(* CODESYS project cy-023_B_PLC1-ifm-206 (AF Logistic Principale).project

Project tree, tasks and I/O mapping:
  AC14nn : AC14nn, ifm electronic, order no. AC14nn, version 3.5.3.002
    application Application
      libraries: ACnnnn_Utils, * (ifm electronic); Standard, * (System); Util, * (System); SysRtc23, 3.4.0.0 (System); SysSocket23, 3.5.4.10 (System); SysFile, 3.5.6.0 (System); SysTypes Interfaces, * (System); CmpErrors Interfaces, * (System); VisuDialogs, * (System); SysFileAsync, 3.5.5.0 (System); NETWORK, 1.2.1.0 (OSCAT)
      task MainTask (cyclic, interval t#20ms, priority 15) calls PLC_PRG
      task EventTask (cyclic, interval t#20ms, priority 5) calls PLC_RT
      task VISU_TASK (cyclic, interval t#200ms, priority 30) calls VisuElems.Visu_Prg
      visualisation VIS_CHONOEDITOR
      visualisation PLC_FileManager
      visualisation PLC_Visualization
    ASi_Master_1 : ASi Master 1, ifm electronic, version 3.5.3.002
      ASi_1_binaryIO : ASi_1_binaryIO, ifm ecomatic gmbh, version 3.5.3.002
          input  Application.PSG_LIST[61] : BOOL  // ASi Input bin.Digital S(A) Slave.Digital S(A) Slave.Bit0
          input  Application.PSG_LIST[62] : BOOL  // ASi Input bin.Digital S(A) Slave.Digital S(A) Slave.Bit2
          input  Application.PSG_LIST[63] : BOOL  // ASi Input bin.Digital S(A) Slave.Digital S(A) Slave.Bit0
          input  Application.PSG_LIST[64] : BOOL  // ASi Input bin.Digital S(A) Slave.Digital S(A) Slave.Bit2
          input  Application.PSG_LIST[65] : BOOL  // ASi Input bin.Digital S(A) Slave.Digital S(A) Slave.Bit0
          input  Application.PSG_LIST[66] : BOOL  // ASi Input bin.Digital S(A) Slave.Digital S(A) Slave.Bit2
          input  Application.PSG_LIST[67] : BOOL  // ASi Input bin.Digital S(A) Slave.Digital S(A) Slave.Bit0
          input  Application.PSG_LIST[68] : BOOL  // ASi Input bin.Digital S(A) Slave.Digital S(A) Slave.Bit2
          input  Application.PSG_LIST[69] : BOOL  // ASi Input bin.Digital S(A) Slave.Digital S(A) Slave.Bit0
          input  Application.PSG_LIST[70] : BOOL  // ASi Input bin.Digital S(A) Slave.Digital S(A) Slave.Bit2
          input  Application.PSG_LIST[71] : BOOL  // ASi Input bin.Digital S(A) Slave.Digital S(A) Slave.Bit0
          input  Application.PSG_LIST[72] : BOOL  // ASi Input bin.Digital S(A) Slave.Digital S(A) Slave.Bit2
          input  Application.PSG_LIST[73] : BOOL  // ASi Input bin.Digital S(A) Slave.Digital S(A) Slave.Bit0
          input  Application.PSG_LIST[74] : BOOL  // ASi Input bin.Digital S(A) Slave.Digital S(A) Slave.Bit2
          input  Application.PSG_LIST[75] : BOOL  // ASi Input bin.Digital S(A) Slave.Digital S(A) Slave.Bit0
          input  Application.PSG_LIST[76] : BOOL  // ASi Input bin.Digital S(A) Slave.Digital S(A) Slave.Bit2
          input  Application.PSG_LIST[77] : BOOL  // ASi Input bin.Digital S(A) Slave.Digital S(A) Slave.Bit0
          input  Application.PSG_LIST[78] : BOOL  // ASi Input bin.Digital S(A) Slave.Digital S(A) Slave.Bit2
          input  Application.PSG_LIST[79] : BOOL  // ASi Input bin.Digital S(A) Slave.Digital S(A) Slave.Bit0
          input  Application.PSG_LIST[80] : BOOL  // ASi Input bin.Digital S(A) Slave.Digital S(A) Slave.Bit2
          input  Application.PSG_LIST[81] : BOOL  // ASi Input bin.Digital S(A) Slave.Digital S(A) Slave.Bit0
          input  Application.PSG_LIST[82] : BOOL  // ASi Input bin.Digital S(A) Slave.Digital S(A) Slave.Bit2
          input  Application.PSG_LIST[83] : BOOL  // ASi Input bin.Digital S(A) Slave.Digital S(A) Slave.Bit0
          input  Application.PSG_LIST[84] : BOOL  // ASi Input bin.Digital S(A) Slave.Digital S(A) Slave.Bit2
          input  Application.PSG_LIST[85] : BOOL  // ASi Input bin.Digital S(A) Slave.Digital S(A) Slave.Bit0
          input  Application.PSG_LIST[86] : BOOL  // ASi Input bin.Digital S(A) Slave.Digital S(A) Slave.Bit2
          input  Application.PSG_LIST[87] : BOOL  // ASi Input bin.Digital S(A) Slave.Digital S(A) Slave.Bit0
          input  Application.PSG_LIST[88] : BOOL  // ASi Input bin.Digital S(A) Slave.Digital S(A) Slave.Bit2
          input  Application.PSG_LIST[121] : BOOL  // ASi Input bin.Digital S(A) Slave.Digital S(A) Slave.Bit0
          input  Application.PSG_LIST[122] : BOOL  // ASi Input bin.Digital S(A) Slave.Digital S(A) Slave.Bit2
          input  Application.PSG_LIST[123] : BOOL  // ASi Input bin.Digital S(A) Slave.Digital S(A) Slave.Bit0
          input  Application.PSG_LIST[124] : BOOL  // ASi Input bin.Digital S(A) Slave.Digital S(A) Slave.Bit2
          input  Application.PSG_LIST[125] : BOOL  // ASi Input bin.Digital S(A) Slave.Digital S(A) Slave.Bit0
          input  Application.PSG_LIST[126] : BOOL  // ASi Input bin.Digital S(A) Slave.Digital S(A) Slave.Bit2
          input  Application.PSG_LIST[127] : BOOL  // ASi Input bin.Digital S(A) Slave.Digital S(A) Slave.Bit0
          input  Application.PSG_LIST[128] : BOOL  // ASi Input bin.Digital S(A) Slave.Digital S(A) Slave.Bit2
          input  Application.PSG_LIST[129] : BOOL  // ASi Input bin.Digital S(A) Slave.Digital S(A) Slave.Bit0
          input  Application.PSG_LIST[130] : BOOL  // ASi Input bin.Digital S(A) Slave.Digital S(A) Slave.Bit2
          input  Application.PSG_LIST[131] : BOOL  // ASi Input bin.Digital S(A) Slave.Digital S(A) Slave.Bit0
          input  Application.PSG_LIST[132] : BOOL  // ASi Input bin.Digital S(A) Slave.Digital S(A) Slave.Bit2
          input  Application.PSG_LIST[133] : BOOL  // ASi Input bin.Digital S(A) Slave.Digital S(A) Slave.Bit0
          input  Application.PSG_LIST[134] : BOOL  // ASi Input bin.Digital S(A) Slave.Digital S(A) Slave.Bit2
          input  Application.PSG_LIST[135] : BOOL  // ASi Input bin.Digital S(A) Slave.Digital S(A) Slave.Bit0
          input  Application.PSG_LIST[136] : BOOL  // ASi Input bin.Digital S(A) Slave.Digital S(A) Slave.Bit2
          input  Application.PSG_LIST[137] : BOOL  // ASi Input bin.Digital S(A) Slave.Digital S(A) Slave.Bit0
          input  Application.PSG_LIST[138] : BOOL  // ASi Input bin.Digital S(A) Slave.Digital S(A) Slave.Bit2
          input  Application.PSG_LIST[139] : BOOL  // ASi Input bin.Digital S(A) Slave.Digital S(A) Slave.Bit0
          input  Application.PSG_LIST[140] : BOOL  // ASi Input bin.Digital S(A) Slave.Digital S(A) Slave.Bit2
          input  Application.PSG_LIST[141] : BOOL  // ASi Input bin.Digital S(A) Slave.Digital S(A) Slave.Bit0
          input  Application.PSG_LIST[142] : BOOL  // ASi Input bin.Digital S(A) Slave.Digital S(A) Slave.Bit2
          input  Application.PSG_LIST[143] : BOOL  // ASi Input bin.Digital S(A) Slave.Digital S(A) Slave.Bit0
          input  Application.PSG_LIST[144] : BOOL  // ASi Input bin.Digital S(A) Slave.Digital S(A) Slave.Bit2
          input  Application.PSG_LIST[145] : BOOL  // ASi Input bin.Digital S(A) Slave.Digital S(A) Slave.Bit0
          input  Application.PSG_LIST[146] : BOOL  // ASi Input bin.Digital S(A) Slave.Digital S(A) Slave.Bit2
          input  Application.PSG_LIST[147] : BOOL  // ASi Input bin.Digital S(A) Slave.Digital S(A) Slave.Bit0
          input  Application.PSG_LIST[148] : BOOL  // ASi Input bin.Digital S(A) Slave.Digital S(A) Slave.Bit2
          input  Application.LUX_ST[43] : BOOL  // ASi Input bin.Digital S(A) Slave.Digital S(A) Slave.Bit0
          input  Application.PSG_LIST[174] : BOOL  // ASi Input bin.Digital S(A) Slave.Digital S(A) Slave.Bit2
          input  Application.LUX_ST[44] : BOOL  // ASi Input bin.Digital S(A) Slave.Digital S(A) Slave.Bit0
          input  Application.PSG_LIST[176] : BOOL  // ASi Input bin.Digital S(A) Slave.Digital S(A) Slave.Bit2
          input  Application.LUX_ST[45] : BOOL  // ASi Input bin.Digital S(A) Slave.Digital S(A) Slave.Bit0
          input  Application.PSG_LIST[178] : BOOL  // ASi Input bin.Digital S(A) Slave.Digital S(A) Slave.Bit2
          input  Application.PSG_LIST[179] : BOOL  // ASi Input bin.Digital B Slave.Digital B Slave.Bit0
          input  Application.PSG_LIST[180] : BOOL  // ASi Input bin.Digital B Slave.Digital B Slave.Bit2
          input  Application.LUX_ST[46] : BOOL  // ASi Input bin.Digital B Slave.Digital B Slave.Bit0
          input  Application.LUX_ST[47] : BOOL  // ASi Input bin.Digital B Slave.Digital B Slave.Bit0
          input  Application.LUX_ST[48] : BOOL  // ASi Input bin.Digital B Slave.Digital B Slave.Bit0
          output Application.LUX_LIST[43] : BOOL  // ASi Output bin.Digital S(A) Slave.Digital S(A) Slave.Bit0
          output Application.LUX_LIST[44] : BOOL  // ASi Output bin.Digital S(A) Slave.Digital S(A) Slave.Bit0
          output Application.LUX_LIST[45] : BOOL  // ASi Output bin.Digital S(A) Slave.Digital S(A) Slave.Bit0
          output Application.LUX_LIST[46] : BOOL  // ASi Output bin.Digital B Slave.Digital B Slave.Bit0
          output Application.LUX_LIST[47] : BOOL  // ASi Output bin.Digital B Slave.Digital B Slave.Bit0
          output Application.LUX_LIST[48] : BOOL  // ASi Output bin.Digital B Slave.Digital B Slave.Bit0
          unmapped channels: ASi Input bin, ASi Output bin
      ASi_1_analogIO : ASi_1_analogIO, ifm ecomatic gmbh, version 3.5.3.002
          unmapped channels: ASi Input, ASi Output
    ASi_Master_2 : ASi Master 2, ifm electronic, version 3.5.3.002
      ASi_2_binaryIO : ASi_2_binaryIO, ifm ecomatic gmbh, version 3.5.3.002
          input  Application.PSG_LIST[1] : BOOL  // ASi Input bin.Digital S(A) Slave.Digital S(A) Slave.Bit0
          input  Application.PSG_LIST[2] : BOOL  // ASi Input bin.Digital S(A) Slave.Digital S(A) Slave.Bit2
          input  Application.PSG_LIST[3] : BOOL  // ASi Input bin.Digital S(A) Slave.Digital S(A) Slave.Bit0
          input  Application.PSG_LIST[4] : BOOL  // ASi Input bin.Digital S(A) Slave.Digital S(A) Slave.Bit2
          input  Application.PSG_LIST[5] : BOOL  // ASi Input bin.Digital S(A) Slave.Digital S(A) Slave.Bit0
          input  Application.PSG_LIST[6] : BOOL  // ASi Input bin.Digital S(A) Slave.Digital S(A) Slave.Bit2
          input  Application.PSG_LIST[7] : BOOL  // ASi Input bin.Digital S(A) Slave.Digital S(A) Slave.Bit0
          input  Application.PSG_LIST[8] : BOOL  // ASi Input bin.Digital S(A) Slave.Digital S(A) Slave.Bit2
          input  Application.PSG_LIST[9] : BOOL  // ASi Input bin.Digital S(A) Slave.Digital S(A) Slave.Bit0
          input  Application.PSG_LIST[10] : BOOL  // ASi Input bin.Digital S(A) Slave.Digital S(A) Slave.Bit2
          input  Application.PSG_LIST[11] : BOOL  // ASi Input bin.Digital S(A) Slave.Digital S(A) Slave.Bit0
          input  Application.PSG_LIST[12] : BOOL  // ASi Input bin.Digital S(A) Slave.Digital S(A) Slave.Bit2
          input  Application.PSG_LIST[13] : BOOL  // ASi Input bin.Digital S(A) Slave.Digital S(A) Slave.Bit0
          input  Application.PSG_LIST[14] : BOOL  // ASi Input bin.Digital S(A) Slave.Digital S(A) Slave.Bit2
          input  Application.PSG_LIST[15] : BOOL  // ASi Input bin.Digital S(A) Slave.Digital S(A) Slave.Bit0
          input  Application.PSG_LIST[16] : BOOL  // ASi Input bin.Digital S(A) Slave.Digital S(A) Slave.Bit2
          input  Application.PSG_LIST[17] : BOOL  // ASi Input bin.Digital S(A) Slave.Digital S(A) Slave.Bit0
          input  Application.PSG_LIST[18] : BOOL  // ASi Input bin.Digital S(A) Slave.Digital S(A) Slave.Bit2
          input  Application.PSG_LIST[19] : BOOL  // ASi Input bin.Digital S(A) Slave.Digital S(A) Slave.Bit0
          input  Application.PSG_LIST[20] : BOOL  // ASi Input bin.Digital S(A) Slave.Digital S(A) Slave.Bit2
          input  Application.PSG_LIST[21] : BOOL  // ASi Input bin.Digital S(A) Slave.Digital S(A) Slave.Bit0
          input  Application.PSG_LIST[22] : BOOL  // ASi Input bin.Digital S(A) Slave.Digital S(A) Slave.Bit2
          input  Application.PSG_LIST[23] : BOOL  // ASi Input bin.Digital S(A) Slave.Digital S(A) Slave.Bit0
          input  Application.PSG_LIST[24] : BOOL  // ASi Input bin.Digital S(A) Slave.Digital S(A) Slave.Bit2
          input  Application.PSG_LIST[25] : BOOL  // ASi Input bin.Digital S(A) Slave.Digital S(A) Slave.Bit0
          input  Application.PSG_LIST[26] : BOOL  // ASi Input bin.Digital S(A) Slave.Digital S(A) Slave.Bit2
          input  Application.PSG_LIST[27] : BOOL  // ASi Input bin.Digital S(A) Slave.Digital S(A) Slave.Bit0
          input  Application.PSG_LIST[28] : BOOL  // ASi Input bin.Digital S(A) Slave.Digital S(A) Slave.Bit2
          input  Application.PSG_LIST[181] : BOOL  // ASi Input bin.Digital S(A) Slave.Digital S(A) Slave.Bit0
          input  Application.PSG_LIST[182] : BOOL  // ASi Input bin.Digital S(A) Slave.Digital S(A) Slave.Bit2
          input  Application.PSG_LIST[183] : BOOL  // ASi Input bin.Digital S(A) Slave.Digital S(A) Slave.Bit0
          input  Application.PSG_LIST[184] : BOOL  // ASi Input bin.Digital S(A) Slave.Digital S(A) Slave.Bit2
          input  Application.PSG_LIST[185] : BOOL  // ASi Input bin.Digital S(A) Slave.Digital S(A) Slave.Bit0
          input  Application.PSG_LIST[186] : BOOL  // ASi Input bin.Digital S(A) Slave.Digital S(A) Slave.Bit2
          input  Application.PSG_LIST[187] : BOOL  // ASi Input bin.Digital S(A) Slave.Digital S(A) Slave.Bit0
          input  Application.PSG_LIST[188] : BOOL  // ASi Input bin.Digital S(A) Slave.Digital S(A) Slave.Bit2
          input  Application.PSG_LIST[189] : BOOL  // ASi Input bin.Digital S(A) Slave.Digital S(A) Slave.Bit0
          input  Application.PSG_LIST[190] : BOOL  // ASi Input bin.Digital S(A) Slave.Digital S(A) Slave.Bit2
          input  Application.PSG_LIST[191] : BOOL  // ASi Input bin.Digital S(A) Slave.Digital S(A) Slave.Bit0
          input  Application.PSG_LIST[192] : BOOL  // ASi Input bin.Digital S(A) Slave.Digital S(A) Slave.Bit2
          input  Application.PSG_LIST[193] : BOOL  // ASi Input bin.Digital S(A) Slave.Digital S(A) Slave.Bit0
          input  Application.PSG_LIST[194] : BOOL  // ASi Input bin.Digital S(A) Slave.Digital S(A) Slave.Bit2
          input  Application.PSG_LIST[195] : BOOL  // ASi Input bin.Digital S(A) Slave.Digital S(A) Slave.Bit0
          input  Application.PSG_LIST[196] : BOOL  // ASi Input bin.Digital S(A) Slave.Digital S(A) Slave.Bit2
          input  Application.PSG_LIST[197] : BOOL  // ASi Input bin.Digital S(A) Slave.Digital S(A) Slave.Bit0
          input  Application.PSG_LIST[198] : BOOL  // ASi Input bin.Digital S(A) Slave.Digital S(A) Slave.Bit2
          input  Application.PSG_LIST[199] : BOOL  // ASi Input bin.Digital S(A) Slave.Digital S(A) Slave.Bit0
          input  Application.PSG_LIST[200] : BOOL  // ASi Input bin.Digital S(A) Slave.Digital S(A) Slave.Bit2
          input  Application.PSG_LIST[201] : BOOL  // ASi Input bin.Digital S(A) Slave.Digital S(A) Slave.Bit0
          input  Application.PSG_LIST[202] : BOOL  // ASi Input bin.Digital S(A) Slave.Digital S(A) Slave.Bit2
          input  Application.PSG_LIST[203] : BOOL  // ASi Input bin.Digital S(A) Slave.Digital S(A) Slave.Bit0
          input  Application.PSG_LIST[204] : BOOL  // ASi Input bin.Digital S(A) Slave.Digital S(A) Slave.Bit2
          input  Application.PSG_LIST[205] : BOOL  // ASi Input bin.Digital S(A) Slave.Digital S(A) Slave.Bit0
          input  Application.PSG_LIST[206] : BOOL  // ASi Input bin.Digital S(A) Slave.Digital S(A) Slave.Bit2
          input  Application.PSG_LIST[207] : BOOL  // ASi Input bin.Digital S(A) Slave.Digital S(A) Slave.Bit0
          input  Application.PSG_LIST[208] : BOOL  // ASi Input bin.Digital S(A) Slave.Digital S(A) Slave.Bit2
          input  Application.LUX_ST[01] : BOOL  // ASi Input bin.Digital S(A) Slave.Digital S(A) Slave.Bit0
          input  Application.LUX_ST[02] : BOOL  // ASi Input bin.Digital S(A) Slave.Digital S(A) Slave.Bit1
          input  Application.PSG_LIST[234] : BOOL  // ASi Input bin.Digital S(A) Slave.Digital S(A) Slave.Bit2
          input  Application.LUX_ST[03] : BOOL  // ASi Input bin.Digital S(A) Slave.Digital S(A) Slave.Bit0
          input  Application.LUX_ST[04] : BOOL  // ASi Input bin.Digital S(A) Slave.Digital S(A) Slave.Bit1
          input  Application.PSG_LIST[236] : BOOL  // ASi Input bin.Digital S(A) Slave.Digital S(A) Slave.Bit2
          input  Application.LUX_ST[05] : BOOL  // ASi Input bin.Digital S(A) Slave.Digital S(A) Slave.Bit0
          input  Application.LUX_ST[06] : BOOL  // ASi Input bin.Digital S(A) Slave.Digital S(A) Slave.Bit1
          input  Application.PSG_LIST[238] : BOOL  // ASi Input bin.Digital S(A) Slave.Digital S(A) Slave.Bit2
          input  Application.LUX_ST[13] : BOOL  // ASi Input bin.Digital B Slave.Digital B Slave.Bit0
          input  Application.LUX_ST[14] : BOOL  // ASi Input bin.Digital B Slave.Digital B Slave.Bit1
          input  Application.PSG_LIST[240] : BOOL  // ASi Input bin.Digital B Slave.Digital B Slave.Bit2
          input  Application.LUX_ST[15] : BOOL  // ASi Input bin.Digital B Slave.Digital B Slave.Bit0
          input  Application.LUX_ST[16] : BOOL  // ASi Input bin.Digital B Slave.Digital B Slave.Bit1
          input  Application.LUX_ST[17] : BOOL  // ASi Input bin.Digital B Slave.Digital B Slave.Bit0
          input  Application.LUX_ST[18] : BOOL  // ASi Input bin.Digital B Slave.Digital B Slave.Bit1
          input  Application.LUX_ST[19] : BOOL  // ASi Input bin.Digital B Slave.Digital B Slave.Bit0
          input  Application.LUX_ST[20] : BOOL  // ASi Input bin.Digital B Slave.Digital B Slave.Bit1
          input  Application.LUX_ST[21] : BOOL  // ASi Input bin.Digital B Slave.Digital B Slave.Bit0
          input  Application.LUX_ST[22] : BOOL  // ASi Input bin.Digital B Slave.Digital B Slave.Bit1
          input  Application.LUX_ST[23] : BOOL  // ASi Input bin.Digital B Slave.Digital B Slave.Bit0
          input  Application.LUX_ST[24] : BOOL  // ASi Input bin.Digital B Slave.Digital B Slave.Bit1
          input  Application.LUX_ST[25] : BOOL  // ASi Input bin.Digital B Slave.Digital B Slave.Bit0
          input  Application.LUX_ST[26] : BOOL  // ASi Input bin.Digital B Slave.Digital B Slave.Bit1
          input  Application.LUX_ST[49] : BOOL  // ASi Input bin.Digital B Slave.Digital B Slave.Bit0
          input  Application.LUX_ST[50] : BOOL  // ASi Input bin.Digital B Slave.Digital B Slave.Bit1
          input  Application.LUX_ST[51] : BOOL  // ASi Input bin.Digital B Slave.Digital B Slave.Bit2
          input  Application.LUX_ST[52] : BOOL  // ASi Input bin.Digital B Slave.Digital B Slave.Bit3
          input  Application.LUX_ST[53] : BOOL  // ASi Input bin.Digital B Slave.Digital B Slave.Bit0
          input  Application.LUX_ST[54] : BOOL  // ASi Input bin.Digital B Slave.Digital B Slave.Bit1
          input  Application.LUX_ST[55] : BOOL  // ASi Input bin.Digital B Slave.Digital B Slave.Bit2
          input  Application.LUX_ST[56] : BOOL  // ASi Input bin.Digital B Slave.Digital B Slave.Bit3
          input  Application.LUX_ST[57] : BOOL  // ASi Input bin.Digital B Slave.Digital B Slave.Bit0
          input  Application.LUX_ST[58] : BOOL  // ASi Input bin.Digital B Slave.Digital B Slave.Bit1
          input  Application.LUX_ST[59] : BOOL  // ASi Input bin.Digital B Slave.Digital B Slave.Bit2
          input  Application.LUX_ST[60] : BOOL  // ASi Input bin.Digital B Slave.Digital B Slave.Bit3
          input  Application.LUX_ST[61] : BOOL  // ASi Input bin.Digital B Slave.Digital B Slave.Bit0
          input  Application.LUX_ST[62] : BOOL  // ASi Input bin.Digital B Slave.Digital B Slave.Bit1
          input  Application.LUX_ST[63] : BOOL  // ASi Input bin.Digital B Slave.Digital B Slave.Bit2
          input  Application.LUX_ST[64] : BOOL  // ASi Input bin.Digital B Slave.Digital B Slave.Bit3
          input  Application.LUX_ST[65] : BOOL  // ASi Input bin.Digital B Slave.Digital B Slave.Bit0
          input  Application.LUX_ST[66] : BOOL  // ASi Input bin.Digital B Slave.Digital B Slave.Bit1
          input  Application.LUX_ST[67] : BOOL  // ASi Input bin.Digital B Slave.Digital B Slave.Bit2
          input  Application.LUX_ST[68] : BOOL  // ASi Input bin.Digital B Slave.Digital B Slave.Bit3
          input  Application.LUX_ST[69] : BOOL  // ASi Input bin.Digital B Slave.Digital B Slave.Bit0
          input  Application.LUX_ST[70] : BOOL  // ASi Input bin.Digital B Slave.Digital B Slave.Bit1
          input  Application.LUX_ST[71] : BOOL  // ASi Input bin.Digital B Slave.Digital B Slave.Bit2
          input  Application.LUX_ST[72] : BOOL  // ASi Input bin.Digital B Slave.Digital B Slave.Bit3
          input  Application.LUX_ST[73] : BOOL  // ASi Input bin.Digital B Slave.Digital B Slave.Bit0
          input  Application.LUX_ST[74] : BOOL  // ASi Input bin.Digital B Slave.Digital B Slave.Bit1
          input  Application.LUX_ST[75] : BOOL  // ASi Input bin.Digital B Slave.Digital B Slave.Bit2
          input  Application.LUX_ST[76] : BOOL  // ASi Input bin.Digital B Slave.Digital B Slave.Bit3
          input  Application.LUX_ST[77] : BOOL  // ASi Input bin.Digital B Slave.Digital B Slave.Bit0
          input  Application.LUX_ST[78] : BOOL  // ASi Input bin.Digital B Slave.Digital B Slave.Bit1
          input  Application.LUX_ST[79] : BOOL  // ASi Input bin.Digital B Slave.Digital B Slave.Bit2
          input  Application.LUX_ST[80] : BOOL  // ASi Input bin.Digital B Slave.Digital B Slave.Bit3
          input  Application.LUX_ST[81] : BOOL  // ASi Input bin.Digital B Slave.Digital B Slave.Bit0
          input  Application.LUX_ST[82] : BOOL  // ASi Input bin.Digital B Slave.Digital B Slave.Bit1
          input  Application.LUX_ST[83] : BOOL  // ASi Input bin.Digital B Slave.Digital B Slave.Bit2
          input  Application.LUX_ST[84] : BOOL  // ASi Input bin.Digital B Slave.Digital B Slave.Bit3
          input  Application.LUX_ST[85] : BOOL  // ASi Input bin.Digital B Slave.Digital B Slave.Bit0
          input  Application.LUX_ST[86] : BOOL  // ASi Input bin.Digital B Slave.Digital B Slave.Bit1
          input  Application.LUX_ST[87] : BOOL  // ASi Input bin.Digital B Slave.Digital B Slave.Bit2
          input  Application.LUX_ST[88] : BOOL  // ASi Input bin.Digital B Slave.Digital B Slave.Bit3
          input  Application.LUX_ST[89] : BOOL  // ASi Input bin.Digital B Slave.Digital B Slave.Bit0
          input  Application.LUX_ST[90] : BOOL  // ASi Input bin.Digital B Slave.Digital B Slave.Bit1
          input  Application.LUX_ST[91] : BOOL  // ASi Input bin.Digital B Slave.Digital B Slave.Bit2
          input  Application.LUX_ST[92] : BOOL  // ASi Input bin.Digital B Slave.Digital B Slave.Bit3
          input  Application.LUX_ST[93] : BOOL  // ASi Input bin.Digital B Slave.Digital B Slave.Bit0
          input  Application.LUX_ST[94] : BOOL  // ASi Input bin.Digital B Slave.Digital B Slave.Bit1
          input  Application.LUX_ST[95] : BOOL  // ASi Input bin.Digital B Slave.Digital B Slave.Bit2
          input  Application.LUX_ST[96] : BOOL  // ASi Input bin.Digital B Slave.Digital B Slave.Bit3
          input  Application.LUX_ST[97] : BOOL  // ASi Input bin.Digital B Slave.Digital B Slave.Bit0
          input  Application.LUX_ST[98] : BOOL  // ASi Input bin.Digital B Slave.Digital B Slave.Bit1
          input  Application.LUX_ST[99] : BOOL  // ASi Input bin.Digital B Slave.Digital B Slave.Bit2
          input  Application.LUX_ST[100] : BOOL  // ASi Input bin.Digital B Slave.Digital B Slave.Bit3
          input  Application.LUX_ST[101] : BOOL  // ASi Input bin.Digital B Slave.Digital B Slave.Bit0
          input  Application.LUX_ST[102] : BOOL  // ASi Input bin.Digital B Slave.Digital B Slave.Bit1
          input  Application.LUX_ST[103] : BOOL  // ASi Input bin.Digital B Slave.Digital B Slave.Bit2
          input  Application.LUX_ST[104] : BOOL  // ASi Input bin.Digital B Slave.Digital B Slave.Bit3
          input  Application.LUX_ST[141] : BOOL  // ASi Input bin.Digital B Slave.Digital B Slave.Bit0
          input  Application.LUX_ST[142] : BOOL  // ASi Input bin.Digital B Slave.Digital B Slave.Bit1
          input  Application.LUX_ST[143] : BOOL  // ASi Input bin.Digital B Slave.Digital B Slave.Bit2
          input  Application.LUX_ST[144] : BOOL  // ASi Input bin.Digital B Slave.Digital B Slave.Bit3
          input  Application.LUX_ST[145] : BOOL  // ASi Input bin.Digital B Slave.Digital B Slave.Bit0
          input  Application.LUX_ST[146] : BOOL  // ASi Input bin.Digital B Slave.Digital B Slave.Bit1
          input  Application.LUX_ST[147] : BOOL  // ASi Input bin.Digital B Slave.Digital B Slave.Bit2
          input  Application.LUX_ST[148] : BOOL  // ASi Input bin.Digital B Slave.Digital B Slave.Bit3
          input  Application.LUX_ST[149] : BOOL  // ASi Input bin.Digital B Slave.Digital B Slave.Bit0
          input  Application.LUX_ST[150] : BOOL  // ASi Input bin.Digital B Slave.Digital B Slave.Bit1
          input  Application.LUX_ST[151] : BOOL  // ASi Input bin.Digital B Slave.Digital B Slave.Bit2
          input  Application.LUX_ST[152] : BOOL  // ASi Input bin.Digital B Slave.Digital B Slave.Bit3
          input  Application.LUX_ST[153] : BOOL  // ASi Input bin.Digital B Slave.Digital B Slave.Bit0
          input  Application.LUX_ST[154] : BOOL  // ASi Input bin.Digital B Slave.Digital B Slave.Bit1
          input  Application.LUX_ST[155] : BOOL  // ASi Input bin.Digital B Slave.Digital B Slave.Bit2
          input  Application.LUX_ST[156] : BOOL  // ASi Input bin.Digital B Slave.Digital B Slave.Bit3
          input  Application.LUX_ST[157] : BOOL  // ASi Input bin.Digital B Slave.Digital B Slave.Bit0
          input  Application.LUX_ST[158] : BOOL  // ASi Input bin.Digital B Slave.Digital B Slave.Bit1
          input  Application.LUX_ST[159] : BOOL  // ASi Input bin.Digital B Slave.Digital B Slave.Bit2
          input  Application.LUX_ST[160] : BOOL  // ASi Input bin.Digital B Slave.Digital B Slave.Bit3
          input  Application.LUX_ST[161] : BOOL  // ASi Input bin.Digital B Slave.Digital B Slave.Bit0
          input  Application.LUX_ST[162] : BOOL  // ASi Input bin.Digital B Slave.Digital B Slave.Bit1
          input  Application.LUX_ST[163] : BOOL  // ASi Input bin.Digital B Slave.Digital B Slave.Bit2
          input  Application.LUX_ST[164] : BOOL  // ASi Input bin.Digital B Slave.Digital B Slave.Bit3
          input  Application.LUX_ST[165] : BOOL  // ASi Input bin.Digital B Slave.Digital B Slave.Bit0
          input  Application.LUX_ST[166] : BOOL  // ASi Input bin.Digital B Slave.Digital B Slave.Bit1
          input  Application.LUX_ST[167] : BOOL  // ASi Input bin.Digital B Slave.Digital B Slave.Bit2
          input  Application.LUX_ST[168] : BOOL  // ASi Input bin.Digital B Slave.Digital B Slave.Bit3
          output Application.LUX_LIST[01] : BOOL  // ASi Output bin.Digital S(A) Slave.Digital S(A) Slave.Bit0
          output Application.LUX_LIST[02] : BOOL  // ASi Output bin.Digital S(A) Slave.Digital S(A) Slave.Bit1
          output Application.LUX_LIST[03] : BOOL  // ASi Output bin.Digital S(A) Slave.Digital S(A) Slave.Bit0
          output Application.LUX_LIST[04] : BOOL  // ASi Output bin.Digital S(A) Slave.Digital S(A) Slave.Bit1
          output Application.LUX_LIST[05] : BOOL  // ASi Output bin.Digital S(A) Slave.Digital S(A) Slave.Bit0
          output Application.LUX_LIST[06] : BOOL  // ASi Output bin.Digital S(A) Slave.Digital S(A) Slave.Bit1
          output Application.LUX_LIST[13] : BOOL  // ASi Output bin.Digital B Slave.Digital B Slave.Bit0
          output Application.LUX_LIST[14] : BOOL  // ASi Output bin.Digital B Slave.Digital B Slave.Bit1
          output Application.LUX_LIST[15] : BOOL  // ASi Output bin.Digital B Slave.Digital B Slave.Bit0
          output Application.LUX_LIST[16] : BOOL  // ASi Output bin.Digital B Slave.Digital B Slave.Bit1
          output Application.LUX_LIST[17] : BOOL  // ASi Output bin.Digital B Slave.Digital B Slave.Bit0
          output Application.LUX_LIST[18] : BOOL  // ASi Output bin.Digital B Slave.Digital B Slave.Bit1
          output Application.LUX_LIST[19] : BOOL  // ASi Output bin.Digital B Slave.Digital B Slave.Bit0
          output Application.LUX_LIST[20] : BOOL  // ASi Output bin.Digital B Slave.Digital B Slave.Bit1
          output Application.LUX_LIST[21] : BOOL  // ASi Output bin.Digital B Slave.Digital B Slave.Bit0
          output Application.LUX_LIST[22] : BOOL  // ASi Output bin.Digital B Slave.Digital B Slave.Bit1
          output Application.LUX_LIST[23] : BOOL  // ASi Output bin.Digital B Slave.Digital B Slave.Bit0
          output Application.LUX_LIST[24] : BOOL  // ASi Output bin.Digital B Slave.Digital B Slave.Bit1
          output Application.LUX_LIST[25] : BOOL  // ASi Output bin.Digital B Slave.Digital B Slave.Bit0
          output Application.LUX_LIST[26] : BOOL  // ASi Output bin.Digital B Slave.Digital B Slave.Bit1
          output Application.LUX_LIST[49] : BOOL  // ASi Output bin.Digital B Slave.Digital B Slave.Bit0
          output Application.LUX_LIST[50] : BOOL  // ASi Output bin.Digital B Slave.Digital B Slave.Bit1
          output Application.LUX_LIST[51] : BOOL  // ASi Output bin.Digital B Slave.Digital B Slave.Bit2
          output Application.LUX_LIST[52] : BOOL  // ASi Output bin.Digital B Slave.Digital B Slave.Bit3
          output Application.LUX_LIST[53] : BOOL  // ASi Output bin.Digital B Slave.Digital B Slave.Bit0
          output Application.LUX_LIST[54] : BOOL  // ASi Output bin.Digital B Slave.Digital B Slave.Bit1
          output Application.LUX_LIST[55] : BOOL  // ASi Output bin.Digital B Slave.Digital B Slave.Bit2
          output Application.LUX_LIST[56] : BOOL  // ASi Output bin.Digital B Slave.Digital B Slave.Bit3
          output Application.LUX_LIST[57] : BOOL  // ASi Output bin.Digital B Slave.Digital B Slave.Bit0
          output Application.LUX_LIST[58] : BOOL  // ASi Output bin.Digital B Slave.Digital B Slave.Bit1
          output Application.LUX_LIST[59] : BOOL  // ASi Output bin.Digital B Slave.Digital B Slave.Bit2
          output Application.LUX_LIST[60] : BOOL  // ASi Output bin.Digital B Slave.Digital B Slave.Bit3
          output Application.LUX_LIST[61] : BOOL  // ASi Output bin.Digital B Slave.Digital B Slave.Bit0
          output Application.LUX_LIST[62] : BOOL  // ASi Output bin.Digital B Slave.Digital B Slave.Bit1
          output Application.LUX_LIST[63] : BOOL  // ASi Output bin.Digital B Slave.Digital B Slave.Bit2
          output Application.LUX_LIST[64] : BOOL  // ASi Output bin.Digital B Slave.Digital B Slave.Bit3
          output Application.LUX_LIST[65] : BOOL  // ASi Output bin.Digital B Slave.Digital B Slave.Bit0
          output Application.LUX_LIST[66] : BOOL  // ASi Output bin.Digital B Slave.Digital B Slave.Bit1
          output Application.LUX_LIST[67] : BOOL  // ASi Output bin.Digital B Slave.Digital B Slave.Bit2
          output Application.LUX_LIST[68] : BOOL  // ASi Output bin.Digital B Slave.Digital B Slave.Bit3
          output Application.LUX_LIST[69] : BOOL  // ASi Output bin.Digital B Slave.Digital B Slave.Bit0
          output Application.LUX_LIST[70] : BOOL  // ASi Output bin.Digital B Slave.Digital B Slave.Bit1
          output Application.LUX_LIST[71] : BOOL  // ASi Output bin.Digital B Slave.Digital B Slave.Bit2
          output Application.LUX_LIST[72] : BOOL  // ASi Output bin.Digital B Slave.Digital B Slave.Bit3
          output Application.LUX_LIST[73] : BOOL  // ASi Output bin.Digital B Slave.Digital B Slave.Bit0
          output Application.LUX_LIST[74] : BOOL  // ASi Output bin.Digital B Slave.Digital B Slave.Bit1
          output Application.LUX_LIST[75] : BOOL  // ASi Output bin.Digital B Slave.Digital B Slave.Bit2
          output Application.LUX_LIST[76] : BOOL  // ASi Output bin.Digital B Slave.Digital B Slave.Bit3
          output Application.LUX_LIST[77] : BOOL  // ASi Output bin.Digital B Slave.Digital B Slave.Bit0
          output Application.LUX_LIST[78] : BOOL  // ASi Output bin.Digital B Slave.Digital B Slave.Bit1
          output Application.LUX_LIST[79] : BOOL  // ASi Output bin.Digital B Slave.Digital B Slave.Bit2
          output Application.LUX_LIST[80] : BOOL  // ASi Output bin.Digital B Slave.Digital B Slave.Bit3
          output Application.LUX_LIST[81] : BOOL  // ASi Output bin.Digital B Slave.Digital B Slave.Bit0
          output Application.LUX_LIST[82] : BOOL  // ASi Output bin.Digital B Slave.Digital B Slave.Bit1
          output Application.LUX_LIST[83] : BOOL  // ASi Output bin.Digital B Slave.Digital B Slave.Bit2
          output Application.LUX_LIST[84] : BOOL  // ASi Output bin.Digital B Slave.Digital B Slave.Bit3
          output Application.LUX_LIST[85] : BOOL  // ASi Output bin.Digital B Slave.Digital B Slave.Bit0
          output Application.LUX_LIST[86] : BOOL  // ASi Output bin.Digital B Slave.Digital B Slave.Bit1
          output Application.LUX_LIST[87] : BOOL  // ASi Output bin.Digital B Slave.Digital B Slave.Bit2
          output Application.LUX_LIST[88] : BOOL  // ASi Output bin.Digital B Slave.Digital B Slave.Bit3
          output Application.LUX_LIST[89] : BOOL  // ASi Output bin.Digital B Slave.Digital B Slave.Bit0
          output Application.LUX_LIST[90] : BOOL  // ASi Output bin.Digital B Slave.Digital B Slave.Bit1
          output Application.LUX_LIST[91] : BOOL  // ASi Output bin.Digital B Slave.Digital B Slave.Bit2
          output Application.LUX_LIST[92] : BOOL  // ASi Output bin.Digital B Slave.Digital B Slave.Bit3
          output Application.LUX_LIST[93] : BOOL  // ASi Output bin.Digital B Slave.Digital B Slave.Bit0
          output Application.LUX_LIST[94] : BOOL  // ASi Output bin.Digital B Slave.Digital B Slave.Bit1
          output Application.LUX_LIST[95] : BOOL  // ASi Output bin.Digital B Slave.Digital B Slave.Bit2
          output Application.LUX_LIST[96] : BOOL  // ASi Output bin.Digital B Slave.Digital B Slave.Bit3
          output Application.LUX_LIST[97] : BOOL  // ASi Output bin.Digital B Slave.Digital B Slave.Bit0
          output Application.LUX_LIST[98] : BOOL  // ASi Output bin.Digital B Slave.Digital B Slave.Bit1
          output Application.LUX_LIST[99] : BOOL  // ASi Output bin.Digital B Slave.Digital B Slave.Bit2
          output Application.LUX_LIST[100] : BOOL  // ASi Output bin.Digital B Slave.Digital B Slave.Bit3
          output Application.LUX_LIST[101] : BOOL  // ASi Output bin.Digital B Slave.Digital B Slave.Bit0
          output Application.LUX_LIST[102] : BOOL  // ASi Output bin.Digital B Slave.Digital B Slave.Bit1
          output Application.LUX_LIST[103] : BOOL  // ASi Output bin.Digital B Slave.Digital B Slave.Bit2
          output Application.LUX_LIST[104] : BOOL  // ASi Output bin.Digital B Slave.Digital B Slave.Bit3
          output Application.LUX_LIST[141] : BOOL  // ASi Output bin.Digital B Slave.Digital B Slave.Bit0
          output Application.LUX_LIST[142] : BOOL  // ASi Output bin.Digital B Slave.Digital B Slave.Bit1
          output Application.LUX_LIST[143] : BOOL  // ASi Output bin.Digital B Slave.Digital B Slave.Bit2
          output Application.LUX_LIST[144] : BOOL  // ASi Output bin.Digital B Slave.Digital B Slave.Bit3
          output Application.LUX_LIST[145] : BOOL  // ASi Output bin.Digital B Slave.Digital B Slave.Bit0
          output Application.LUX_LIST[146] : BOOL  // ASi Output bin.Digital B Slave.Digital B Slave.Bit1
          output Application.LUX_LIST[147] : BOOL  // ASi Output bin.Digital B Slave.Digital B Slave.Bit2
          output Application.LUX_LIST[148] : BOOL  // ASi Output bin.Digital B Slave.Digital B Slave.Bit3
          output Application.LUX_LIST[149] : BOOL  // ASi Output bin.Digital B Slave.Digital B Slave.Bit0
          output Application.LUX_LIST[150] : BOOL  // ASi Output bin.Digital B Slave.Digital B Slave.Bit1
          output Application.LUX_LIST[151] : BOOL  // ASi Output bin.Digital B Slave.Digital B Slave.Bit2
          output Application.LUX_LIST[152] : BOOL  // ASi Output bin.Digital B Slave.Digital B Slave.Bit3
          output Application.LUX_LIST[153] : BOOL  // ASi Output bin.Digital B Slave.Digital B Slave.Bit0
          output Application.LUX_LIST[154] : BOOL  // ASi Output bin.Digital B Slave.Digital B Slave.Bit1
          output Application.LUX_LIST[155] : BOOL  // ASi Output bin.Digital B Slave.Digital B Slave.Bit2
          output Application.LUX_LIST[156] : BOOL  // ASi Output bin.Digital B Slave.Digital B Slave.Bit3
          output Application.LUX_LIST[157] : BOOL  // ASi Output bin.Digital B Slave.Digital B Slave.Bit0
          output Application.LUX_LIST[158] : BOOL  // ASi Output bin.Digital B Slave.Digital B Slave.Bit1
          output Application.LUX_LIST[159] : BOOL  // ASi Output bin.Digital B Slave.Digital B Slave.Bit2
          output Application.LUX_LIST[160] : BOOL  // ASi Output bin.Digital B Slave.Digital B Slave.Bit3
          output Application.LUX_LIST[161] : BOOL  // ASi Output bin.Digital B Slave.Digital B Slave.Bit0
          output Application.LUX_LIST[162] : BOOL  // ASi Output bin.Digital B Slave.Digital B Slave.Bit1
          output Application.LUX_LIST[163] : BOOL  // ASi Output bin.Digital B Slave.Digital B Slave.Bit2
          output Application.LUX_LIST[164] : BOOL  // ASi Output bin.Digital B Slave.Digital B Slave.Bit3
          output Application.LUX_LIST[165] : BOOL  // ASi Output bin.Digital B Slave.Digital B Slave.Bit0
          output Application.LUX_LIST[166] : BOOL  // ASi Output bin.Digital B Slave.Digital B Slave.Bit1
          output Application.LUX_LIST[167] : BOOL  // ASi Output bin.Digital B Slave.Digital B Slave.Bit2
          output Application.LUX_LIST[168] : BOOL  // ASi Output bin.Digital B Slave.Digital B Slave.Bit3
          unmapped channels: ASi Input bin, ASi Output bin
      ASi_2_analogIO : ASi_2_analogIO, ifm ecomatic gmbh, version 3.5.3.002
          unmapped channels: ASi Input, ASi Output
    Fieldbus_Interface : Fieldbus Interface, ifm electronic, version 3.5.3.002
      FieldBusData_ : FieldBusData  , ifm ecomatic gmbh, version 3.5.3.002
          unmapped channels: Inputs from fieldbus, Outputs to fieldbus
      ASi_1_binaryOut : ASi_1_binaryOut, ifm ecomatic gmbh, version 3.5.3.002
          unmapped channels: FB ASi Output bin
      ASi_1_analogOut : ASi_1_analogOut, ifm ecomatic gmbh, version 3.5.3.002
          unmapped channels: FB ASi Output ana
      ASi_2_binaryOut : ASi_2_binaryOut, ifm ecomatic gmbh, version 3.5.3.002
          unmapped channels: FB ASi Output bin
      ASi_2_analogOut : ASi_2_analogOut, ifm ecomatic gmbh, version 3.5.3.002
          unmapped channels: FB ASi Output ana
    Ethernet : Ethernet, ifm electronic, version 3.4.2.0
  Utils Functions/
    function ADDSTRING [ST]
    function block AVERAGE_DINT [ST]: Read, Reset
    function block AVERAGE_INT [ST]: Read, Reset
    function block AVERAGE_T [ST]: Read, Reset
    function CHKSTRING [ST]
    function COPY_32SWAP16 [ST]
    function DWORDSWAP [ST]
    function block FLT_EVENT [ST]
    function block FLT_TAP [ST]
    function block FLT_TIME [ST]
    function HEXTORAW [ST]
    function LINEAR [ST]
    function LINEAR_BAD [ST]
    function MEMCLR [ST]
    function MEMCPY [ST]
    function block DELAYRETRY [ST]: Start, Success, Fail
    function RAW16TOHEXSTR [ST]
    function RAWTOHEX [ST]
    function RAWTOHEXSTR [ST]
    function STR_NOSPACES [ST]
    function block TCPCLIENT [ST]
    function block TCPSERVER [ST]
    function block TONOF [ST]
    function ADR_AT_INT [ST]
    function block TestAsi_FB [ST]
    function AsiInMapping [ST]
    function AsiOutMapping [ST]
    function block OpenFiles_ASI_PSG_FB [ST]
    function GenerateTabs [ST]
    function block OpenFiles_ASI_LUX_FB [ST]
    function block OpenFiles_ASI_PSG_FB_backup [ST]
    function block OpenFiles_LUX_PSG_FB [ST]
    function block OpenFiles_Default_LUX_FB [ST]
    function block FileCopyToSD_FB [ST]
    function block FileCopySDToPLC_FB [ST]
    function block LuxEnable_FB [ST]
    function block LuxTimerModify_FB [ST]
    function block LuxManOnOff_FB [ST]
    function block OpenFiles_CFG_FB [ST]
    function block DirOpen_FB [ST]
    function block FileSize_and_Time_FB [ST]
    SysDirAsync
  Plant_obj/
    function block obj_ASI [ST]
    function block obj_CRON [ST]: DB_Create, DB_Load, DB_SetName, Init, AddLogData
    function block obj_CRON_EDITOR [ST]: CA_Load_Exe, CA_Save_Exe, FileOpen, JL_Load_Exe, JL_Save_Exe, PR_Load_Exe, PR_Save_Exe
    function block obj_LUXM [ST]: AddLogData, StatReset
    function block obj_PSG [ST]: StatReset, AddLogData
    function block obj_PSG_old [ST]: StatReset
    function block obj_LUXM_old [ST]: AddLogData, StatReset
    function block obj_LUXM_backUp [ST]: AddLogData, StatReset
  Utils/
    function CSV_Log [ST]
    function RTC_Update [ST]
  TCP_Logger/
    function LogEv [ST]
    function Logger_Head [ST]
    program Logger_Proc [ST]: MsgChk, MsgSave
    function Logger_Send [ST]
    function LogTrig [ST]
  TCP_Remote/
    program Remote_Proc [ST]: Cmd_CAL, Cmd_CRON, Cmd_GRU, Cmd_PDC, Cmd_SYS, Command, Cmd_LUX
  _Variables/
    global variables Global_Constants
    global variables Global_Retain
    global variables Global_Variables
  _Datatypes/
    Logger/
      data type en_Logger_ErrLev
      data type en_Logger_Status
      data type typ_Logger
      data type en_Logger_Sel
    data type en_SYS_Objects
    data type en_SYS_Status
    data type typ_SYS
    Plant_Objects/
      data type typ_Cron_Calendar
      data type typ_Cron_Jolly
      data type typ_Cron_Profile
    data type type_TabAsiPsg
    data type type_TabAsiLux
    data type type_TabLuxPsg
    data type type_TabDefaultLux
    data type type_DataLuxForVis
    data type type_TabCfg
    data type type_DataPsgForVis
    data type en_RotGrun
    data type type_AsiOutput
  program PLC_PRG [ST]: MainCtrl
  program PLC_RT [ST]
  text list GlobalTextList
*)

// _Datatypes/Logger/en_Logger_ErrLev
TYPE en_Logger_ErrLev :
(
	EL_Log			:=0,
	EL_Wrn			:=1,
	EL_Alarm		:=2,
	EL_AlarmStop	:=3
);
END_TYPE

// _Datatypes/Logger/en_Logger_Status
TYPE en_Logger_Status :
(
	S_Logger_UNKNOWN := 0,
	S_Logger_IDLE,
	S_Logger_WAITCONN,
	S_Logger_WAITTX,
	S_Logger_WAITRESP,
	S_Logger_ERROR
);
END_TYPE

// _Datatypes/Logger/typ_Logger
TYPE typ_Logger :
STRUCT
	Status		: en_Logger_Status;

	SendReq		: BOOL;
	SendIdx		: DWORD;
	SendData	: ARRAY [0..MAX_SEND_TCP_CLIENT] OF BYTE;
	SendLen		: DWORD;	//DINT; GIURE ver 4

	TData		: ARRAY [0..MAX_SEND_TCP_CLIENT] OF BYTE;
	TLen		: DWORD;	//DINT; GIURE ver 4

	LastIdxPos	: DWORD;

	(* Temporary variables used by objects *)
	s1			: STRING(256);
	i1			: WORD;

END_STRUCT
END_TYPE

// _Datatypes/en_SYS_Objects
TYPE en_SYS_Objects :
(
	EO_SYS		:=0,  (* PLC *)
	EO_VPN		:=1,  (* VPN *)
	EO_DOOR		:=2,  (* Door & access control *)

	EO_CAL		:=10, (* Caldaia *)
	EO_CIR		:=11, (* Circolatore *)
	EO_CRON		:=12, (* Crono-termostato *)
	EO_VRD		:=13, (* Valvola miscelatore pannelli *)
	EO_CTL		:=14, (* Contalitri *)
	EO_CTB		:=15, (* Contabilizzatore *)
	EO_TPV		:=16, (* Temperature probes values *)
	EO_PPV		:=17, (* Pressure probes values *)
	EO_PBV		:=18, (* Over-Pressure Alarms *)
	EO_TBV		:=19, (* Over-Temperature Alarms *)
	EO_PMV		:=20, (* Under-Pressure Alarms *)
	EO_GRU		:=21, (* Gruppo termico *)
	EO_PDC		:=22, (* Pompa di calore *)
	EO_SOL		:=23, (* Pannello solare termico *)
	EO_ESOL		:=24, (* Pannello solare fotovoltaico *)
	EO_GAS		:=25, (* Contatore GAS *)
	EO_PORT		:=26, (* Misuratore di portata *)
	EO_FPV		:=27, (* Flow probes values *)
	EO_ANZ		:=28, (* Analizzatore di rete *)
	EO_SCA		:=29, (* Signal Control Alarms *)
	EO_LUX		:=30, (* Base Illumination point *)
	EO_LUXM		:=31, (* Metered Illumination point *)
	EO_PSG		:=32, (* Sensore di passaggio *)
	EO_HVAC		:=33, (* Heating, Ventilating and Air Conditioning *)
	EO_HYGRV	:=34, (* Relative Humidity sensors value *)
	EO_COOV		:=35, (* Carbon Dioxide CO2 sensors value *)

	EO_ZGW			:=200,  (* ZigBee - Gateway *)
	EO_ZRM			:=201,	(* ZigBee - Repeater *)
	EO_ZREL			:=202,	(* ZigBee - Actuator rele *)
	EO_ZTHL			:=203,	(* ZigBee - Temperature Sensor *)

	EO_ASGW			:=250,	(* ASi - Gateway *)
	EO_ASCBI		:=251,	(* ASi - Input Board, Ciabatta *)

	EO_LON			:=1000, (* Bus - LON *)
	EO_MODBUS		:=1001, (* Bus - MODBUS *)
	EO_MBUS			:=1002, (* Bus - M-BUS *)
	EO_MODBUS_TCP	:=1003, (* Bus - MODBUS TCP *)

	EO_GENERIC		:=9000, (* Generic dataset *)
	EO_EXPO			:=9001  (* EXPO dataset *)
);
END_TYPE

// _Datatypes/en_SYS_Status
TYPE en_SYS_Status :
(
	S_UNKNOWN  := 0,
	S_STARTUP,
	S_INIT_RTC,
	S_INIT_VAR,
	S_AUTOTEST,
	S_RUNNING,
	S_SHUTDOWN,
	S_HALT,
	S_RELOAD
);
END_TYPE

// _Datatypes/typ_SYS
TYPE typ_SYS :
STRUCT
	Status			: en_SYS_Status;
	Warning			: BOOL;
	Alarm			: BOOL;
	AlarmStop		: BOOL;

	Time_LogString	: STRING;
	Time_Year		: WORD;
	Time_Month		: BYTE;
	Time_Day		: BYTE;
	Time_Hour		: BYTE;
	Time_Min		: BYTE;

	Time_CT_DT		: DT;
	Time_CT_Day		: WORD;
	Time_CT_Quarter	: BYTE;

	LastLogs_Idx	: BYTE;
	LastLogs_Dat	: ARRAY[0..5] OF STRING;
	LastLogs_Msg	: ARRAY[0..5] OF STRING;

END_STRUCT
END_TYPE

// _Datatypes/Plant_Objects/typ_Cron_Calendar
TYPE typ_Cron_Calendar :
STRUCT
	Profile		: ARRAY[0..384] OF BYTE;
END_STRUCT
END_TYPE

// _Datatypes/Plant_Objects/typ_Cron_Jolly
TYPE typ_Cron_Jolly :
STRUCT
	Start		: DT;
	End			: DT;
	Temp		: INT;
	Flags		: WORD; (* B0:Enabled B1..B15:Unused *)
END_STRUCT
END_TYPE

// _Datatypes/Plant_Objects/typ_Cron_Profile
TYPE typ_Cron_Profile :
STRUCT
	Flags		: WORD;
	Setpoint	: ARRAY [0..95] OF INT;
END_STRUCT
END_TYPE

// _Datatypes/type_TabAsiPsg
TYPE type_TabAsiPsg :
STRUCT
	Asi1_2: BYTE;
	Address: BYTE;
	A_B: BYTE;
	bit_psg	: ARRAY [0..MAX_BIT] OF WORD;
END_STRUCT
END_TYPE

(*
TYPE type_TabAsiPsg :
STRUCT
	Asi1_2: BYTE;
	Address: BYTE;
	A_B: BYTE;
	Bit_address : BYTE;
	PSG: WORD;
END_STRUCT
END_TYPE
*)

// _Datatypes/type_TabAsiLux
TYPE type_TabAsiLux :
STRUCT
	Asi1_2: BYTE;
	Address: BYTE;
	A_B: BYTE;
	bit_lux	: ARRAY [0..MAX_BIT] OF WORD;
END_STRUCT
END_TYPE
(*
TYPE type_TabAsiLux :
STRUCT
	Asi1_2: BYTE;
	Address: BYTE;
	A_B: BYTE;
	Bit_address : BYTE;
	LUX: WORD;
END_STRUCT
END_TYPE
*)

// _Datatypes/type_TabLuxPsg
TYPE type_TabLuxPsg : 
STRUCT
	LuxId	: WORD; //Id del lux da controllare
	TimerOn	: TIME; //Tempo di accensione del lux
	h_Start	: TOD;	//Orario di start del controllo a timer
	h_End	: TOD;	//Orario di off del controllo a timer
	scaIdUnit	: BYTE; //Componente unità di SCA
	scaIdDec	: BYTE; //Componente decimale di SCA
	PSG_list: ARRAY [0..MAX_PSGLIST] OF WORD; //elenco dei passaggi associati al lux 
END_STRUCT
END_TYPE

// _Datatypes/type_TabDefaultLux
TYPE type_TabDefaultLux :
STRUCT
	LuxNumber: WORD;
	Mode: BYTE;
END_STRUCT
END_TYPE

// _Datatypes/type_DataLuxForVis
//La seguente struttura ha la funzione di collegare l'id del lux con i relativi dati qui indicati
//In tal modo la visualizzazione dello stato dei lux viene eseguita associando l'ID dell'array contenente questa struttura

TYPE type_DataLuxForVis :
STRUCT
	VisStatus	: dword; //valori di status_vis
	VisTimer	: time;	//Valori dei timer
	VisMod		: byte; //Impostazione mode
END_STRUCT
END_TYPE

// _Datatypes/type_TabCfg
type type_TabCfg : 
	struct
		id_Clevergy		: word; //identificativo dell'impianto
		id_Plc			: byte; //identificativo del plc
		HourOfControl	: byte;	//Ora a cui avviene il controllo dello stato dei psg (o altri elementi). Si controlla se i psg sono ok 
		MinOfControl	: byte;	//Minuti a ui avviene il controllo 
		TimeOutError	: TIME; //Tempo allo scadere del quale se il psg è interrotto si genera un allarme (tipico 30 min) 
	end_struct
end_type

// _Datatypes/type_DataPsgForVis
//La seguente struttura ha la funzione di collegare l'id del psg con i relativi dati qui indicati
//In tal modo la visualizzazione dello stato dei psg viene eseguita associando l'ID dell'array contenente questa struttura

TYPE type_DataPsgForVis :
STRUCT
	VisStatus	: dword; //valori di status_vis
END_STRUCT
END_TYPE

// _Datatypes/Logger/en_Logger_Sel
TYPE en_Logger_Sel :
(
	Sel_PSG := 0,
	Sel_LUX := 1,
	Sel_CRON:= 2,
	Sel_END
);
END_TYPE

// _Datatypes/en_RotGrun
TYPE en_RotGrun :
(
	ROT := 0,
	GRUN:= 1
);
END_TYPE

// _Datatypes/type_AsiOutput
TYPE type_AsiOutput :
STRUCT
	AsiDigitalOut:	bool;
	AsiAnalogOut:	word;
END_STRUCT
END_TYPE

// _Variables/Global_Constants
{attribute 'global_init_slot' := '300'}
VAR_GLOBAL CONSTANT
	//PLC_ID		: STRING := '2'; //Identificativo del plc	
	ASI_TOT		: BYTE := 128; //ASI1_A+ASI1_B+ASI2_A+ASI2_B = 32*4=128
	MAX_BIT		: BYTE := 3;
	MAX_ASI		: BYTE := 32;
	MAX_PSGLIST	: BYTE := 9;  //numero massimo di passaggi associati ad ogni lux 0..9
	MAX_LUXNUM	: WORD := 250;	//512; //numero massimo di bit su rete asi (asi1A + asi1B + asi2A + asi2B)* 4 bit = 512. Quindi numero massimo di lux abbinabili alla rete asi completa
	PSG_MAXNUM	: WORD := 250;	//512;
	CRON_MAX	: WORD := 250;	//512;
	
	LUXM_MAX_ID	: WORD := 900; //Numero massimo associabile ad un lux (id del lux)
	PSG_MAX_ID	: WORD := 900; //Numero massimo associabile ad un pasaggio (id del passaggio)
	
	//Dim array retentivi
	MAX_PSG_RETAIN	: BYTE := 250;
	MAX_LUX_RETAIN	: BYTE := 250;
		
	(* Filesystem *)
	LogsPath			: STRING :='/media/sd/';
	ConfPath			: STRING :='/media/sd/';
	MapConf_Path		: STRING :='/media/sd/';
	AsiPsg_FileName		: STRING :='_ASI_PSG.txt';
	AsiLux_FileName		: STRING :='_ASI_LUX.txt';
	LuxPsg_FileName		: STRING :='_AUT_LUX_PSG.txt';
	DefaultLux_FileName	: STRING :='_DEF_LUX.txt';
	Cfg_FileName		: STRING :='CFG.txt';
	//FilesPath			: STRING :='/media/sd/';(*'';*)(*'S:\';*)

	(* Visu colours *)	
	COLOR_RED 		: DWORD:=16#F02020;
	COLOR_YELLOW	: DWORD:=16#F0F020;
	COLOR_GREEN		: DWORD:=16#20F020;
	COLOR_GREEN_OFF : DWORD:=16#108010;
	COLOR_LBLUE		: DWORD:=16#80F0F0;
	COLOR_GREY		: DWORD:=16#C0C0C0;
	
	(******************************************************)
	(**************** MOVE OUTSIDE HERE *******************)
	(* TCP Logger *)
	Logger_SERVER		: STRING:='';
	Logger_IP			: STRING:='178.33.227.41';//'10.88.32.183'; //'192.168.100.3';
	Logger_PORT			: WORD  :=80;
//	Logger_GETSTART		: STRING:='GET /cygmsrv/AFLgm.ashx?';
//	Logger_GETEND		: STRING:='$R$N$R$N';
//	Logger_CHECK		: STRING:='True';
	Logger_CRLF			: STRING:='$R$N';
	Logger_DataFile		: STRING:='/media/sd/LOG.DAT';
	Logger_DataFileOld	: STRING:='/media/sd/LOG.BCK';
	Logger_IndexFile	: STRING:='/media/sd/LOG.IDX';
	Logger_ConnRetries	: BYTE:=5;
	Logger_RecoverMsgs	: BYTE:=50;
	(* TCP Remote *)
	Remote_PORT			: WORD  :=10;
	Remote_WELCOME		: STRING:='Connected$R$N';
	(* TCP Sockets *)
	MAX_SEND_TCP_SERVER					 : DWORD:=1500;(*60000*)
	MAX_RECEIVE_TCP_SERVER				 : WORD:=3000;	//DWORD:=3000; GIURE ver 206
	MAX_RECEIVE_TCP_SERVER_SOCKET	 	 : DWORD:=1500;
	MAX_SEND_TCP_CLIENT					 : DWORD:=4096;(*15000*)
	MAX_RECEIVE_TCP_CLIENT				 : DWORD:=1500;
	MAX_RECEIVE_TCP_CLIENT_SOCKET		 : DWORD:=1500;
	MAX_RECEIVE_UDP_SERVER				 : INT  :=1472;
	MAX_RECEIVE_UDP_CLIENT				 : INT  :=1472;
	CONNECT_WATCHDOG_TIME				 : TIME :=T#10S;
	(******************************************************)
	ASI_A	: BYTE:=0;
	ASI_B	: BYTE:=1;
END_VAR

// _Variables/Global_Retain
VAR_GLOBAL RETAIN
	Mode_Manual : BOOL := FALSE;

	PsgCounter		: ARRAY [1..MAX_PSG_RETAIN] OF WORD;

//	WORKINGTIME		: ARRAY [1..LUXM_MAX] OF DWORD; (* [sec] Internal working time counter *)
//	POWERONCYCLES	: ARRAY [1..LUXM_MAX] OF DWORD; (* Internal counter of power-on cycles *)
//	ENERGYCOUNTER	: ARRAY [1..LUXM_MAX] OF DWORD; (* [E-1 kWh] Internal energy counter *)
//	ENERGYCOUNTER_T : ARRAY [1..LUXM_MAX] OF DWORD; (* Temporary energy in E-2*Wsec *)

	WORKINGTIME_n	: ARRAY [1..MAX_LUX_RETAIN] OF DWORD; (* [sec] Internal working time counter *)
	POWERONCYCLES_n	: ARRAY [1..MAX_LUX_RETAIN] OF word;	//DWORD; (* Internal counter of power-on cycles *)
	ENERGYCOUNTER_n	: ARRAY [1..MAX_LUX_RETAIN] OF word; //DWORD; (* [E-1 kWh] Internal energy counter *)
	ENERGYCOUNTER_T_n : ARRAY [1..MAX_LUX_RETAIN] OF DWORD; (* Temporary energy in E-2*Wsec *)
	
END_VAR

// _Variables/Global_Variables
VAR_GLOBAL
	Plant_NAME			: STRING :='cySN:xx cyVER:03 - AF-Logistics Principale';	//NON MODIFICARE PRIMA DEL CARATTERE '-'	
	Plant_SN			: DWORD;  //:=23;	 	// S/N Impianto di telecontrollo. Viene rilevato dal file cfg.txt
	PLC_ID				: STRING; //:= '2'; //Identificativo del plc - interno al file cfg.txt	
	Plant_SW_VER		: WORD   :=03;		// Versione SW installata. 
//	ControlTime			: TIME_OF_DAY;		//variabile di controllo orario
	
	SYS    : typ_SYS;
	Logger : typ_Logger;
	CronEd : obj_CRON_EDITOR;

	(**** PLANT OBJECTS ****)
	ASI01: obj_ASI				:=( ID:=1 );
	ASI02: obj_ASI				:=( ID:=2 );

	PSG		: ARRAY [1..PSG_MAXNUM] OF obj_PSG;
	
	CRON   : ARRAY [1..CRON_MAX] OF obj_CRON;
	
	ptPSG : POINTER TO obj_PSG;

	ptLUX : POINTER TO obj_LUXM;
	LuxVar, LuxVar2 : obj_LUXM;

	TabAsiPsg	: ARRAY [1..ASI_TOT] OF type_TabAsiPsg; //Mappa di lettura dati provenienti dal file ASI_PSG
	TabASILux	: ARRAY [1..ASI_TOT] OF type_TabAsiLux; //Mappa di lettura dati provenienti dal file ASI_LUX
	TabLuxPsg	: ARRAY [1..MAX_LUXNUM] OF type_TabLuxPsg; //Tabella contenente l'elenco dei lux automatici e dei relativi passaggi che li azionano
	TabDefaultLux : ARRAY [1..MAX_LUXNUM] OF type_TabDefaultLux; //Tabella dei valori di default dei lux, ovvero 
	TabCfg		: type_TabCfg;	//Dati letti da cfg.txt
															//lux --> 00:Man off, 01:Man On, 02:Cronografo, 03: Automatico (timer su laser)
	LuxElement	: ARRAY [1..MAX_LUXNUM] OF obj_LUXM;  //Lista di variabili Lux
	DataLuxForVis	: array [1..MAX_LUXNUM] of type_DataLuxForVis;	//Array ordinato contenente i valori Status_Vis e del timer utilizzati per la visualizzazione (PLC_Visualization)
	DataPsgForVis	: array [1..MAX_LUXNUM] of type_DataPsgForVis;	//Array ordinato contenente i valori Status_Vis utilizzati per la visualizzazione (PLC_Visualization)
	
	ASI_1	 : ARRAY [ASI_A..ASI_B,1..MAX_ASI,0..MAX_BIT] OF BOOL; //Mappa asi_1 per monitoraggio input e attuazione output
	ASI_2	 : ARRAY [ASI_A..ASI_B,1..MAX_ASI,0..MAX_BIT] OF BOOL; //Mappa asi_2 per monitoraggio input e attuazione output
	PSG_LIST : ARRAY [1..PSG_MAX_ID] OF BOOL; //900
	LUX_LIST : ARRAY [1..LUXM_MAX_ID] OF BOOL; //900
	LUX_ST	 : ARRAY [1..LUXM_MAX_ID] OF BOOL; //900

	LuxOutput_ASI: ARRAY [1..LUXM_MAX_ID] OF BOOL;	//900 - Variabili settate nei rispettivi LuxElement per essere poi passate alle uscite (LUX_LIST[y]) {7..12=6, 27..42=16, 46..48=3, 105..168=64}
	
	//Gestione SD card
	//SD_Card	: obj_SD;
	
	DirNames: array[1..64] of string;
	FileNames: array[1..64] of string;
	UpDownKey : word := 1;	
	(**** SIMULATION ONLY ****)
	TEST1:BOOL;	
	KEYON:BOOL;
	KEYVIRT:BOOL;
	(*...*)

	Logger_GETSTART		: STRING:='GET /cygmsrv/AFLgm.ashx?';
	Logger_GETEND		: STRING:='$R$N$R$N';
	Logger_CHECK		: STRING:='True';
	
	enSelect			: en_Logger_Sel:= Sel_PSG;
END_VAR

// PLC_PRG
PROGRAM PLC_PRG
VAR
	Timer1	: TON; (* Fast controls tick *)
	Timer2	: TON; (* Plant control tick *)
	Timer3	: TON; (* Logger timer *)
	Timer10 : TON; (* Logger timer delay *)
	i 		: BYTE;
	ValInCrono			:	INT; //Valore del setpoint del crono
	VisLuxOnOffSelected	:	word;//lux selezionato in plc visu per on/off
	TimerLuxSelected	:	word;//lux selezionato in plc visu per modifica timer
	VisValueManAut		: 	bool;//valore del selettore a visualizzazione: 0=manuale 1= automatico (crono)
	VisValueManOnOff	: 	bool;//valore del selettore a visualizzazione valido se il precedente è in manuale: 0=spento 1= acceso 
	
	TestAsi	: TestAsi_FB;
	
	OpenFileASI_PSG 		: OpenFiles_ASI_PSG_FB;
	OpenFileASI_LUX 		: OpenFiles_ASI_LUX_FB;
	OpenFileLUX_PSG 		: OpenFiles_LUX_PSG_FB;
	OpenFiles_Default_LUX 	: OpenFiles_Default_LUX_FB;
	OpenFiles_CFG			: OpenFiles_CFG_FB;
	
	FileCopyToSD	: FileCopyToSD_FB;
	FileCopySDToPLC	: FileCopySDToPLC_FB;
	
	FileSize_and_Time 	: FileSize_and_Time_FB;
	LuxTimerModify	:LuxTimerModify_FB;
	LuxManOnOff		:LuxManOnOff_FB;
	
	TestPSG		: BOOL;
	count		: INT := 0;
	sMapFileName: STRING;
	viewFileName: STRING;
	CopyToSd	: BOOL;
	CopyToPLC	: BOOL;
	MakeDirOpen : BOOL;
	FileTime	: BOOL;
	ReLoadFiles	: BOOL;
	SlideFile	: BOOL;
	VisModify_T_Lux: bool;
	VisModify_Man_Lux : bool;
	TimerLuxValue: dword;
	UpDownKey: word;
	UpKey, DownKey: word;
	counter : WORD;
	LuxCount: WORD;
	PsgCount: BYTE;
	x, j, y	: WORD;
	LocalRefTableLuxPsg: WORD;
	Message		: STRING;
	LogSemaphore: en_RotGrun;
END_VAR

(******************************************************************************
 ****                           MAIN TASK CODE                             ****
 ******************************************************************************

	Network setup: PLC_2
		IP  = 10.88.32.182 | MSK = 255.255.255.0
		GW	= 10.88.32.13 | DNS = //////192.168.100.1
		SNTP = //////193.204.114.232 (3600s) ==> 192.168.100.3

*)
//---------------------------------------------------------------------------//
// GIURE ver 023_002 	AFLogistic_Principale	(04/02/16)
// Versione completa testata e contenente molto codice da ripulire
//---------------------------------------------------------------------------//
//---------------------------------------------------------------------------//
// GIURE ver 023_001 	AFLogistic_Principale
// Versione intermedia con le seguenti funzioni:
// Lettura dei dati provenienti dai file di configurazione presenti sulla SD
// Configurazione corretta della rete asi
// Bozza degli obj_PSG e obj_LUXM
// test con:
//			sensori laser posizionati su indirizzi asi-2 1A bit 0 e bit 2
//			Lux 105 e 107 posizionati su indirizzi asi-2 13B bit 0 e bit 2
//---------------------------------------------------------------------------//

(*==============================*)
(*===== Main status machine ====*)
(*==============================*)
MainCtrl();

(*==============================*)
(*== Running cycle operations ==*)
(*==============================*)
(*
IF SYS.Status>S_INIT_VAR THEN

END_IF
*)
(*==============================*)
(*== System cycle operations ===*)
(*==============================*)
(* Execute TCP processes *)
Logger_Proc();
Remote_Proc();
//Logger_Proc();
//										Remote_Proc();
(* Update user led *)
(*USRLED_Update();*)
(* Execute Cron Editor commands *)
CronEd();
(* External resources *)
(*
   IF NOT TPV01.ERR THEN T_AMB:=T_S01;
ELSIF NOT TPV05.ERR THEN T_AMB:=GRU01.TAmb;
ELSE 					 T_AMB:=Plant_DefaultTAmb;
END_IF
*)
//TestAsi();
(**** SIMULATION ONLY ****)
(*...*)

ACTION MainCtrl:
case Sys.Status of

	S_STARTUP:
		(* Initialize array objects *)
		//open file at startup - Operazioni da ripetere nella sequenza di reload dei files (S_RELOAD)
		OpenFiles_CFG();
		OpenFileASI_PSG();
		OpenFileASI_LUX();
		OpenFileLUX_PSG();
		OpenFiles_Default_LUX();
		j:=0;
		for counter := 1 to MAX_LUXNUM do
			LuxElement[counter].ID := TabDefaultLux[counter].LuxNumber; //copio id del lux nella tabella delle variabili dei lux
			LuxElement[counter].CTRL_MODE := TabDefaultLux[counter].Mode; //copio il mode nella tabella delle variabili dei lux
			LuxElement[counter].CTRL_MODE_backUp := TabDefaultLux[counter].Mode; //salvo il mode di backup per il ripristina modo
			//Se il mode è timer (3) cerco lo stesso ID in TabLuxPsg e pone il valore RefTableAutLuxPsg all'indice a cui si trova x 
			//In pratica RefTableAutLuxPsg linka LuxElement[] a TabLuxPsg[]
			if LuxElement[counter].CTRL_MODE = 3 then
				for x := 1 to MAX_LUXNUM do
					if TabLuxPsg[x].LuxId = LuxElement[counter].ID
						then 
							LuxElement[counter].RefTableAutLuxPsg := x;
							LuxElement[counter].LuxTimer := TabLuxPsg[x].TimerOn; //set del valore del timer del lux
					end_if
				end_for
			end_if
			if LuxElement[counter].CTRL_MODE = 2 then
				j:=j+1;
				CRON[j].ID:=TabDefaultLux[counter].LuxNumber;	
			end_if
		end_for
		
		Sys.Status:=S_INIT_RTC;
	S_INIT_RTC:
		(* Check RTC and update from network *)
		RTC_Update();
		(* Check time *)
		if Sys.Time_Year>2000 then
			Sys.Status:=S_INIT_VAR;
		end_if
	S_INIT_VAR:
		LogEv(EL_Wrn,EO_SYS,0,1,CONCAT('System_1_startup_v',WORD_TO_STRING(Plant_SW_VER)));
		Sys.Status:=S_RUNNING;

	S_RUNNING:
		Timer2(IN:=not Timer2.Q,PT:=T#500MS);
		if Timer2.Q then
			(* Read current date/time *)
			RTC_Update();
		end_if
		if ReLoadFiles then
			Sys.Status:=S_RELOAD;	
			Message:='Reload File request';
			ReLoadFiles := FALSE;
		end_if
		if CopyToSd //Se viene premuto il tasto corrispondente di copia file
			then 
				FileCopyToSD();
				CopyToSd := FALSE;
		end_if
		if CopyToPLC //Se viene premuto il tasto corrispondente di copia file
			then 
				FileCopySDToPLC();
				CopyToPLC := FALSE;
		end_if
		if FileTime
			then
				FileSize_and_Time();
				FileTime := FALSE;
		end_if
			
(*		if MakeDirOpen //Se viene premuto il tasto corrispondente di open directory
			then 
//				DirOpen();
				MakeDirOpen := FALSE;
		end_if *)
		if  SlideFile then
			//viewFileName:=FileNames[UpDownKey];
			
			SlideFile := FALSE;
		end_if
		if VisModify_T_Lux
			then LuxTimerModify(NewValueTimer := TimerLuxValue, IdFind := PLC_PRG.TimerLuxSelected);
				VisModify_T_Lux := FALSE;
		end_if
		if VisModify_Man_Lux
			then LuxManOnOff(NewValueManSw0 := bool_to_byte(VisValueManOnOff), NewValueManSw1 := bool_to_byte(VisValueManAut), IdFind := PLC_PRG.VisLuxOnOffSelected);
				VisModify_Man_Lux := FALSE;
		end_if
		
		ASI01();
		ASI02();
		
		(* External switch *)
		//KEYON:=EXT_KEY1 OR EXT_KEY2 OR EXT_KEY3 OR KEYVIRT;
		LuxCount := 1;
		while LuxElement[LuxCount].ID <> 0 do //esegue scansione dei lux dell'impianto solo se presenti
		//for LuxCount := 1 to MAX_LUXNUM do 
			case LuxElement[LuxCount].CTRL_MODE of
			0: 
				LuxElement[LuxCount](WORKINGTIME:=WORKINGTIME_n[LuxCount], 
														POWERONCYCLES:=POWERONCYCLES_n[LuxCount],
														ENERGYCOUNTER:=ENERGYCOUNTER_n[LuxCount], 
														ENERGYCOUNTER_T:=ENERGYCOUNTER_T_n[LuxCount],
														CtrlExton:=KEYON);
			1: 
				LuxElement[LuxCount](WORKINGTIME:=WORKINGTIME_n[LuxCount], 
														POWERONCYCLES:=POWERONCYCLES_n[LuxCount],
														ENERGYCOUNTER:=ENERGYCOUNTER_n[LuxCount], 
														ENERGYCOUNTER_T:=ENERGYCOUNTER_T_n[LuxCount],
														CtrlExton:=KEYON);
			2: 	//se il mode è settato come cronografo gestisco accensione a orologio
				CRON[LuxCount]( SetPoint=>ValInCrono);
				LuxElement[LuxCount].ValInCronoInLux:=ValInCrono;
				LuxElement[LuxCount](WORKINGTIME:=WORKINGTIME_n[LuxCount], 
														POWERONCYCLES:=POWERONCYCLES_n[LuxCount],
														ENERGYCOUNTER:=ENERGYCOUNTER_n[LuxCount], 
														ENERGYCOUNTER_T:=ENERGYCOUNTER_T_n[LuxCount],
														CtrlExton:=KEYON);
				
			3:  //se il mode è settato come automatico gestisco l'accensione a timer con innesco da sensori laser
					for PsgCount := 0 to MAX_PSGLIST do //all'interno dell'associazione lux passaggi controllo quali passaggi sono presenti
						if TabLuxPsg[LuxElement[LuxCount].RefTableAutLuxPsg].PSG_list[PsgCount]<>0
							then//memorizzo il riferimento alla tabella Lux-Psg in una var locale che userò per indicizzare successivamente
								LocalRefTableLuxPsg := TabLuxPsg[LuxElement[LuxCount].RefTableAutLuxPsg].PSG_list[PsgCount];
								y:=1;
								//Cerco all'interno dell'array dei PSG in quale locazione si trova quello con l'ID memorizzato in LocalRefTableLuxPsg
								while (PSG[y].ID <> LocalRefTableLuxPsg) and (y <= PSG_MAXNUM) do
									y:=y+1;
								end_while
								if PSG[y].ID = LocalRefTableLuxPsg
									then
										LuxElement[LuxCount].CtrlTrig:=PSG[y].xSense_trig;
										LuxElement[LuxCount](WORKINGTIME:=WORKINGTIME_n[LuxCount], 
																				POWERONCYCLES:=POWERONCYCLES_n[LuxCount],
																				ENERGYCOUNTER:=ENERGYCOUNTER_n[LuxCount], 
																				ENERGYCOUNTER_T:=ENERGYCOUNTER_T_n[LuxCount],
																				CtrlExton:=KEYON);
								END_IF
						end_if
					end_for
			end_case
			LuxCount := LuxCount + 1;
		end_while
		Timer3(IN:=NOT Timer3.Q,PT:=T#5m);
		IF Timer3.Q THEN
			LogSemaphore:=GRUN;
			(* Trig logger *)
//			LogTrig();
			(* Execute temporary CSV logger *)
			(*CSV_Log();*)
		END_IF
		if LogSemaphore = GRUN then
			Timer10(IN:=NOT Timer10.Q,PT:=T#15s);
			if Timer10.Q then
				LogTrig();
			end_if
			if enSelect=Sel_END then //La commutazione del valore di enSelect avviene in LogTrig. Corrisponde al restart del log
				LogSemaphore := ROT;
				enSelect:=Sel_PSG;
				Timer10(IN:=TRUE,PT:=T#5s);
			end_if
//			if enSelect=Sel_PSG then //La commutazione del valore di enSelect avviene in LogTrig. Corrisponde al restart del log
//				LogSemaphore := ROT;
//				Timer10(IN:=TRUE,PT:=T#5s);
//			end_if
		end_if	
		
	S_RELOAD:
		OpenFiles_CFG();
		OpenFileASI_PSG();
		OpenFileASI_LUX();
		OpenFileLUX_PSG();
		OpenFiles_Default_LUX();
		j:=0;
		for counter := 1 to MAX_LUXNUM do
			LuxElement[counter].ID := TabDefaultLux[counter].LuxNumber; //copio id del lux nella tabella delle variabili dei lux
			LuxElement[counter].CTRL_MODE := TabDefaultLux[counter].Mode; //copio il mode nella tabella delle variabili dei lux
			//Se il mode è timer (3) cerco lo stesso ID in TabLuxPsg e pone il valore RefTableAutLuxPsg all'indice a cui si trova x 
			//In pratica RefTableAutLuxPsg linka LuxElement[] a TabLuxPsg[]
			if LuxElement[counter].CTRL_MODE = 3 then
				for x := 1 to MAX_LUXNUM do
					if TabLuxPsg[x].LuxId = LuxElement[counter].ID
						then 
							LuxElement[counter].RefTableAutLuxPsg := x;
							LuxElement[counter].LuxTimer := TabLuxPsg[x].TimerOn; //set del valore del timer del lux
					end_if
				end_for
			end_if
			if LuxElement[counter].CTRL_MODE = 2 then
				j:=j+1;
				CRON[j].ID:=TabDefaultLux[counter].LuxNumber;	
			end_if
		end_for
		Message:=' File reloaded';
		LogEv(EL_Wrn,EO_SYS,0,1,CONCAT('System_reload_files',WORD_TO_STRING(Plant_SW_VER)));
		Sys.Status:=S_RUNNING;
	
else
	Sys.Status:=S_STARTUP;
end_case;
END_ACTION

END_PROGRAM

// Plant_obj/obj_PSG
FUNCTION_BLOCK obj_PSG
(* === Passage sensor ===   v1.0[23/12/15] - Giudici R. *)
//Rileva i fronti di salita e discesa dello stato del sensore passaggio e lo meorizza in xSense_trig.
//Il dato viene usato per gestire accensione del lux corrispondente e per controllo errori sul sensore

VAR_INPUT
	(* Settings *)
	ID				: WORD;
	//ptNextPsg, ptPrevPsg : POINTER TO obj_PSG := 16#FFFFFFFF;
	TimErr_timeout	: TIME;	//:=T#30M; (* Timeout for occupied barrier error *)
	TimeOfControl	: TOD;
	TimeString		: STRING;
	EVH_TimeOutError: bool;
	NotifyLog		: bool;
(*	WRN_TIMEOUT		: TIME:=T#5M;  (* Timeout fot occupied barrier warning *)*)	
(*	ACT_TIMEOUT 	: TIME:=T#7D;  (* Timeout for inactive barrier warning *)*)
(*	DISTANCE		: WORD; 	   (* Distance to 2th sensor in mm *)*)
(*  SPEED_THRESHOLD : INT;         (* Speed threshold for output trigger *)*)
	(* Ack output events *)
	//xSense_trig		: BOOL;
	(* Physical inputs *)
	Psg_state	: BOOL;				//Stato del sensore associato al passaggio
(*	PSG_IN2			: BOOL;        (* Optional speed input sensor *)*)	
END_VAR
VAR_IN_OUT
	NumTransition		: WORD;	//numero di transizioni eseguite, max: 16#FFFF
(*	SPEED			: AVERAGE_INT; *)	
END_VAR
VAR_OUTPUT
	xSense_trig		: BOOL;	//set a 1 sul fronte di salita della fotocellula corrispondente
	(* Status *)
	Status_Log		: BYTE;
	Status_Vis 		: DWORD;
END_VAR
VAR
	evnt	: FLT_EVENT;
	errt	: TON;
	errtev	: FLT_EVENT;
	
	TrigH:	BOOL;
	fTrigFun: F_TRIG;
	rTrigFun: R_TRIG;
(*	wrnt	: TON;*)
(*	actt	: TON:*)
END_VAR

TimErr_timeout :=  TabCfg.TimeOutError; //Set del valore del timeout error al valore caricato dal file cfg.txt
//function start
fTrigFun(CLK:=Psg_state);	//rilevo fronte di discesa - raggio infrarosso interrotto
rTrigFun(CLK:=Psg_state);	//rilevo fronte di salita - raggio infrarosso ripristinato
IF fTrigFun.q THEN	// se raggio infrarosso interrotto
	Status_Vis:=COLOR_GREEN; //Vado a popolare la visualizzazione con il verde
	xSense_trig := TRUE;	//memorizzo il fronte di salita
	IF NumTransition=16#FFFF THEN	//16#FFFFFFFF
		LogEv(EL_Wrn,EO_PSG,ID,5,''); //Warning numero passaggi massimi raggiunto - reset contatore
		NumTransition:=1;
	ELSE
		NumTransition:=NumTransition+1;	//incremento contatore transizioni al passaggio
	END_IF
END_IF
IF rTrigFun.q THEN	//se raggio infrarosso ripristinato 
	 xSense_trig := FALSE;	//reset del fronte di salita
END_IF

(* Error check *)
//Il check avviene solo ad un orario giornaliero impostato in cfg.txt e l'allarme viene inoltrato solo se il tempo () di infrarosso interrotto è scaduto
errt(IN:=xSense_trig, PT:=TimErr_timeout);
errtev(IN:=errt.Q);
IF errtev.EVH THEN
	EVH_TimeOutError := TRUE; //posto a true quando scade il timer del check error
	NotifyLog := FALSE;	//posto a true nel momento in cui viene iniltrato il log Event
END_IF

if (EVH_TimeOutError = TRUE) and  (NotifyLog = FALSE) and (TabCfg.HourOfControl = Sys.Time_Hour) and (TabCfg.MinOfControl = Sys.Time_Min)	
	then
		NotifyLog := TRUE;
		Status_Log:=2; Status_Vis:=COLOR_RED;
		LogEv(EL_Alarm,EO_PSG,ID,2,'');	//warning timeout passaggio interrotto
end_if

IF (errtev.EVL) and (EVH_TimeOutError = TRUE) and (NotifyLog = TRUE)
THEN
	NotifyLog := FALSE;
	EVH_TimeOutError := FALSE;
	Status_Log:=0; Status_Vis:=COLOR_GREEN;
	LogEv(EL_Log,EO_PSG,ID,1,''); // passaggio interrotto ripristinato (status OK)
END_IF

//Salvataggio dati in array ordinato per numero di ID utile per la visualizzazione
DataPsgForVis[ID].VisStatus:=Status_Vis;

ACTION StatReset:
(* Reset statistic counters *)
NumTransition:=0;
END_ACTION

ACTION AddLogData:
//Genera la stringa di log dei passaggi	//GIURE ver 23_002

Logger.s1:=INSERT('&PSG=',WORD_TO_STRING(ID),4);
IF ID<10 THEN Logger.s1:=INSERT(Logger.s1,'0',4); END_IF

Logger.s1:=CONCAT(Logger.s1,WORD_TO_STRING(NumTransition));		
Logger.s1:=CONCAT(Logger.s1,';');

ADDSTRING(ADR(Logger.TData), ADR(Logger.s1), Logger.TLen);
END_ACTION

END_FUNCTION_BLOCK

// TCP_Logger/LogEv
FUNCTION LogEv : BOOL
VAR_INPUT
	Level	: en_Logger_ErrLev;
	Object  : en_SYS_Objects;
	Index	: WORD;
	Error	: WORD;
	Message : STRING;
END_VAR
VAR
	s1 : STRING(160);
	i  : INT;
END_VAR

(* Execute error level operations *)
CASE Level OF
	EL_Wrn: 		Sys.Warning:=TRUE;
	EL_Alarm: 		Sys.Alarm  :=TRUE;
	EL_AlarmStop: 	Sys.Alarm  :=TRUE; (* GO TO STOP STATE!! *)
END_CASE

(* Fill lastlog list *)
s1:=CONCAT(Sys.Time_LogString,';Lev=');
s1:=CONCAT(s1,INT_TO_STRING(Level));
s1:=CONCAT(s1,';Obj=');
s1:=CONCAT(s1,INT_TO_STRING(Object));
s1:=CONCAT(s1,';Idx=');
s1:=CONCAT(s1,WORD_TO_STRING(Index));
s1:=CONCAT(s1,';Err=');
s1:=CONCAT(s1,WORD_TO_STRING(Error));
Sys.LastLogs_Dat[Sys.LastLogs_Idx]:=s1;
Sys.LastLogs_Msg[Sys.LastLogs_Idx]:=Message;
Sys.LastLogs_Idx:=Sys.LastLogs_Idx+1;
IF Sys.LastLogs_Idx>5 THEN Sys.LastLogs_Idx:=0; END_IF

(*---------------------------------------------------------------*)
	Logger_Head();
(*---------------------------------------------------------------*)

(* Insert ERR *)
s1:=CONCAT('&ERR=',INT_TO_STRING(Level));
s1:=CONCAT(s1,';');
s1:=CONCAT(s1,INT_TO_STRING(Object));
s1:=CONCAT(s1,';');
s1:=CONCAT(s1,WORD_TO_STRING(Index));
s1:=CONCAT(s1,';');
s1:=CONCAT(s1,WORD_TO_STRING(Error));
s1:=CONCAT(s1,';');
ADDSTRING(ADR(Logger.TData), ADR(s1), Logger.TLen);
s1:=Message;
STR_NOSPACES(ADR(s1));
ADDSTRING(ADR(Logger.TData), ADR(s1), Logger.TLen);

(*---------------------------------------------------------------*)
	Logger_Send();
//	Logger_Send();
(*---------------------------------------------------------------*)

END_FUNCTION

// TCP_Logger/Logger_Head
FUNCTION Logger_Head : BOOL
VAR
	s1 : STRING(160);
	i  : BYTE;
END_VAR

Logger.TLen:=0;
(* Set GET header *)
ADDSTRING(ADR(Logger.TData), ADR(Logger_GETSTART), Logger.TLen);

(* Insert Header *)
//s1:=INSERT('ID=&V=&D=',DWORD_TO_STRING(Plant_SW_VER),6);
//s1:=INSERT(s1,DWORD_TO_STRING(Plant_SN),3);
s1:=INSERT('ID=&V=1&D=',DWORD_TO_STRING(Plant_SN),3);
s1:=CONCAT(s1,Sys.Time_LogString);
s1:=CONCAT(s1,'&S=');
IF Sys.Alarm THEN i:=2; ELSIF Sys.Warning THEN i:=1; ELSE i:=0; END_IF
s1:=CONCAT(s1,BYTE_TO_STRING(i));
ADDSTRING(ADR(Logger.TData), ADR(s1), Logger.TLen);

END_FUNCTION

// Utils Functions/ADDSTRING
FUNCTION ADDSTRING : BOOL (* Append string to a byte buffer *)
VAR_INPUT
	pTxData: POINTER TO BYTE;
	pString: POINTER TO BYTE;
END_VAR
VAR_IN_OUT
	TxLen: DWORD;	//DINT;
END_VAR
VAR
END_VAR

pTxData:=pTxData+TxLen;
WHILE pString^<>0 DO
	pTxData^:=pString^;
	pString:=pString+1;
	pTxData:=pTxData+1;
	TxLen:=TxLen+1;
END_WHILE

END_FUNCTION

// Utils Functions/STR_NOSPACES
FUNCTION STR_NOSPACES : BOOL (* Replace spaces and bad chars with allowed ones, used as HTTP-GET validator *)
VAR_INPUT
	pString: POINTER TO BYTE;
END_VAR
VAR
END_VAR

WHILE pString^<>0 DO
	IF pString^=16#20 (* space *) THEN pString^:=16#5F; (*'_'*) END_IF
	pString:=pString+1;
END_WHILE

END_FUNCTION

// TCP_Logger/Logger_Send
FUNCTION Logger_Send : BOOL
VAR
	hFile		: RTS_IEC_HANDLE;
	hRes		: RTS_IEC_RESULT;
	pos:	DWORD;
	ts: STRING;
	ts2: STRING;
END_VAR

(* Finalize string *)
ADDSTRING(ADR(Logger.TData), ADR(Logger_GETEND), Logger.TLen);

(* Read log position *)
ts:=Logger_DataFile;
pos:=SysFileGetSize(ts, ADR(hRes));
(* Check log size, bckup and erase if no pending messages *)
IF pos>1000000 THEN
	ts:=Logger_IndexFile;
	hFile:=SysFileOpen(ts,AM_READ,ADR(hRes));
	IF hFile=RTS_INVALID_HANDLE THEN
		ts:=Logger_DataFileOld;
		SysFileDelete(ts);
		ts:=Logger_DataFile; ts2:=Logger_DataFileOld;
		SysFileRename(ts,ts2);
		pos:=0;
	ELSE
		SysFileClose(hFile);
	END_IF
END_IF
(* Write message on log file *)
ts:=Logger_DataFile;
hFile:=SysFileOpen(ts,AM_APPEND_PLUS,ADR(hRes));
IF hFile<>RTS_INVALID_HANDLE THEN
	SysFileWrite(hFile, ADR(Logger.TData), Logger.TLen, ADR(hRes));
	SysFileClose(hFile);
ELSE
	Sys.Warning:=TRUE;
END_IF


(* Check logger status *)
IF Logger.SendReq=FALSE THEN
	(* Set log position for recovery *)
	Logger.SendIdx:=pos;
	(* Copy message data *)
	MEMCPY(ADR(Logger.TData),ADR(Logger.SendData),Logger.TLen);
	Logger.SendLen:=Logger.TLen;
	(* Trigger request *)
	Logger.SendReq:=TRUE;
ELSE
	(* Add message position+size in recovery indexes *)
	ts:=Logger_IndexFile;
	hFile:=SysFileOpen(ts, AM_APPEND_PLUS, ADR(hRes));
	SysFileWrite(hFile, ADR(pos), SIZEOF(pos), ADR(hRes));
	SysFileWrite(hFile, ADR(Logger.TLen), SIZEOF(Logger.TLen), ADR(hRes));
	SysFileClose(hFile);
END_IF

END_FUNCTION

// Utils Functions/MEMCPY
FUNCTION MEMCPY:BOOL
VAR_INPUT
	pSourceAddress:POINTER TO ARRAY[1..2] OF BYTE;
	pDestinationAddress:POINTER TO ARRAY[1..2] OF BYTE;
	BytesToCopy:DWORD;	// GIURE ver 4 WORD;
END_VAR
VAR
END_VAR

WHILE (BytesToCopy > 0) DO
	pDestinationAddress^[1]:=pSourceAddress^[1]; (* copy bytes from source to destination *)
	pDestinationAddress:=ADR(pDestinationAddress^[2]); (* increment destination *)
	pSourceAddress:=ADR(pSourceAddress^[2]);(* increment source *)
	BytesToCopy:=BytesToCopy -1; (* decrement number of bytes to copy *)
END_WHILE

END_FUNCTION

// Utils Functions/AVERAGE_INT
FUNCTION_BLOCK AVERAGE_INT
VAR_INPUT
	IN: 	INT;
END_VAR
VAR_OUTPUT
	HI:		INT;
	AVG:	INT;
	LOW:	INT;
	ERR:	BOOL;
END_VAR
VAR
	sum:	DINT;
	cnt:	WORD;
END_VAR

IF cnt>=65000 THEN
	ERR:=TRUE;
	Read();
	sum := sum - AVG;
	cnt := cnt - 1;
END_IF

sum := sum + IN;
cnt := cnt + 1;

IF IN<LOW THEN LOW:=IN; END_IF
IF IN>HI  THEN HI :=IN; END_IF

ACTION Read:
AVG := DINT_TO_INT(sum/cnt);
END_ACTION

ACTION Reset:
HI:=IN;
AVG:=IN;
LOW:=IN;
ERR:=FALSE;

sum:=IN;
cnt:=1;
END_ACTION

END_FUNCTION_BLOCK

// Utils Functions/FLT_EVENT
FUNCTION_BLOCK FLT_EVENT
VAR_INPUT
	IN		: BOOL;
	INITEV	: BOOL:=TRUE;
END_VAR
VAR_OUTPUT
	EVH		: BOOL;
	EVL		: BOOL;
END_VAR
VAR
	init	: BOOL:=FALSE;
	old		: BOOL;
END_VAR

EVH:=FALSE;
EVL:=FALSE;

IF NOT init THEN
	init:=TRUE;
	IF INITEV THEN
		old := NOT IN;
	ELSE
		old := IN;
	END_IF
END_IF

IF old<>IN THEN
	old:=IN;
	IF IN THEN EVH:=TRUE; ELSE EVL:=TRUE; END_IF
END_IF

END_FUNCTION_BLOCK

// Plant_obj/obj_LUXM
FUNCTION_BLOCK obj_LUXM
(* === Metered ON/OFF Illumination Point ===
   Failure detection:
   Statistic data:
   
   - Come identifico l'assenza del nodo?? (Rele non funzionante/non alimentato)
   - Acquisizione carico dopo accensione?? Dati carico in NVM!
   
   v1.0[07/05/15] - Create
   v2.0[jan-2016] - Modify GIURE
*)
VAR_INPUT
	(* Settings *)
	ID				: WORD;
	//ptNextLux, ptPrevLux : POINTER TO obj_LUXM := 16#FFFFFFFF;
	(* Controls *)
	CTRL_MODE		: BYTE;  (* 0:MAN OFF, 1:MAN-ON, 3:Timer laser, 2:Cronografo*)
	CTRL_MODE_backUp: BYTE;
	LuxTimer		: TIME; //Tempo di accensione del lux settato nella tabella TabLuxPsg ottenuta dal file di config su SD
	ValInCronoInLux : INT;	//Valore del setpoint arrivato dal crono
	RefTableAutLuxPsg : WORD; //indice di riferimento alla tabella AUT_LUX_PSG se mode = 3
	CtrlTrig		: BOOL; (* Trigger for timer start *)
	CtrlKey			: BOOL; (* External KEY control input *)
	CtrlSens		: BOOL; (* External dark sensor input [1:Dark] *)
	CtrlExton		: BOOL; (* External forced activation *)
	(* Physical inputs *)
	REL_ST			: BOOL; (* Status feedback *)
	REL_V			: WORD; (* [E-1 V] Voltage *)
	REL_A			: WORD; (* [E-1 A] Current *)
	REL_ALM			: WORD; (* Error status [0:OK, 1:Disconnected, 2:LoadLOW, 3:LoadHIGH, 4:Overload, 5:ControlFAIL] *)
	REL_TEMP		: INT;  (* [E-1 °C] Temperature *)
	REL_TON			: DWORD;(* [sec] External working time counter *)  
	(* Persistent *)
	//PressKeyVisuOn	: BOOL := 0;
	//PressKeyVisuOff	: BOOL := 0;
END_VAR
VAR_IN_OUT
//VAR_OUTPUT RETAIN PERSISTENT
	
	WORKINGTIME		: DWORD; (* [sec] Internal working time counter *)
	POWERONCYCLES	: word;	//DWORD; (* Internal counter of power-on cycles *)
	ENERGYCOUNTER	: word;	//DWORD; (* [E-1 kWh] Internal energy counter *)
	ENERGYCOUNTER_T : DWORD; (* Temporary energy in E-2*Wsec *)
END_VAR
VAR_OUTPUT
	(* Physical outputs *)
	REL_EN			: BOOL;	// uscita logica per compatibilità con sw preesistente (ex (* Control output *))
	(* Status *)
	Status_Log		: BYTE;
	Status_Vis 		: DWORD;
END_VAR
VAR
	TickTimer		: TON := ( PT:=T#1S );
	TrigTimer		: TOF ;
	sREL_EN			: FLT_EVENT;
	sREL_ALM		: WORD:=16#FFFF;
	chkREL_ST		: FLT_TIME := ( TTAP:=T#20S, INITEV:=FALSE );
	
	ModeToServer : byte;
	ForcedOn : byte;
	ForcedOff : byte;	

END_VAR

//---------------- Info sulla logica di controllo --------------------------------//
//Dato che il relè asi controlla un relè NC la logica di controllo è negata, quindi:
//			LuxOutput_ASI[ID] := FALSE; indica Lux acceso 
//			LuxOutput_ASI[ID] := TRUE; indica Lux spento 
//--------------------------------------------------------------------------------//
//Con l'ID si identifica il numero del lux sul campo quindi il suo valore può variare da 1 a LUXM_MAX (attualmente 1...900)
(* Control logic *)
if CtrlExton then	//accensione del lux con controllo manuale
	LuxOutput_ASI[ID] := FALSE; //Lux acceso
else
	case CTRL_MODE of
	0: //Manuale Off
		LuxOutput_ASI[ID] := TRUE;
	1: //Manuale On
		LuxOutput_ASI[ID] := FALSE;
	2: //Cronografo
		if ValInCronoInLux = 1000 //OR ( LuxElement[i].PressKeyVisuOn)
			then
			LuxOutput_ASI[ID] := FALSE; //Lux acceso
			else if ValInCronoInLux = 0 //OR ( NOT LuxElement[i].PressKeyVisuOn)
				then
				LuxOutput_ASI[ID] := TRUE; //Lux spento
			end_if
		end_if
	3: //Timer 
		(* Trig timer *)
		TrigTimer.PT:=LuxTimer;	//TIME_LUX_DEF;
		TrigTimer(IN:= CtrlTrig);
		
		if TrigTimer.Q then 
			LuxOutput_ASI[ID] := FALSE; //Lux acceso
			else
				LuxOutput_ASI[ID] := TRUE; //Lux spento
		end_if
	end_case
end_if

//-----------------------------------------------------------------------------------------------------------
//Se i pin del feedback relè non sono cavallottati si usa la seguente riga al posto di quelle successive indicate da(#)
//REL_ST := LUX_ST[ID];	
//-----------------------------------------------------------------------------------------------------------

//setting della variabile REL_EN per compatibilità con il sw preesistente
if LuxOutput_ASI[ID] = TRUE  //Lux spento
	then	
		REL_ST := FALSE;	//A causa del cavallotto sui pin del relè forzo a falso (#)
		REL_EN := FALSE;
	elsif LuxOutput_ASI[ID] = FALSE  //Lux acceso
		then
			REL_ST := LUX_ST[ID];	//Quando so che la luce è accesa leggo lo stato del pin (che essendo cavallottato sarà a 1) (#)
			REL_EN := TRUE;
end_if
(* Temporary energy counter *)
TickTimer(IN:=not TickTimer.Q);
if TickTimer.Q AND REL_EN then
//if TickTimer.Q and not LuxOutput_ASI[ID] then
	WORKINGTIME:=WORKINGTIME+1;
	ENERGYCOUNTER_T:=ENERGYCOUNTER_T+REL_V*REL_A;
	if ENERGYCOUNTER_T>36000000 then
		ENERGYCOUNTER_T:=ENERGYCOUNTER_T-36000000;
		ENERGYCOUNTER:=ENERGYCOUNTER+1;		
	end_if
end_if

(* Generate status events *)
sREL_EN(IN:=REL_EN);
if sREL_EN.EVL then LogEv(EL_Log,EO_LUX,ID,2,''); end_if
if sREL_EN.EVH then LogEv(EL_Log,EO_LUX,ID,3,''); POWERONCYCLES:=POWERONCYCLES+1; end_if

(* Check status feedback *)
chkREL_ST(IN:=(REL_ST<>REL_EN));
if chkREL_ST.EVH then LogEv(EL_Alarm,EO_LUX,ID,9,''); end_if
if chkREL_ST.EVL AND sREL_ALM=0 then LogEv(EL_Log,EO_LUX,ID,1,''); end_if

(* Check controller alarm *)
if sREL_ALM<>REL_ALM then
	case REL_ALM of
		0: if not chkREL_ST.OUT then LogEv(EL_Log,EO_LUX,ID,1,''); end_if
		1: LogEv(EL_Alarm,EO_LUX,ID,6,'');
		2: LogEv(EL_Wrn  ,EO_LUX,ID,4,WORD_TO_STRING(REL_A));
		3: LogEv(EL_Wrn  ,EO_LUX,ID,5,WORD_TO_STRING(REL_A));
		4: LogEv(EL_Alarm,EO_LUX,ID,7,WORD_TO_STRING(REL_A));
		5: LogEv(EL_Alarm,EO_LUX,ID,8,'');
	end_case
	sREL_ALM:=REL_ALM;
end_if

(* Status color *)
   if REL_ALM=1 OR REL_ALM>3 OR chkREL_ST.OUT	then Status_Log:=2; Status_Vis:=COLOR_RED;
elsif REL_ALM<>0								then Status_Log:=1; Status_Vis:=COLOR_YELLOW;
                  	   							else Status_Log:=0; Status_Vis:=SEL(REL_EN,COLOR_GREEN_OFF,COLOR_GREEN);
end_if

//Salvataggio dati in array ordinato per numero di ID utile per la visualizzazione
DataLuxForVis[ID].VisStatus:=Status_Vis; 
DataLuxForVis[ID].VisTimer:=LuxTimer/1000;	
DataLuxForVis[ID].VisMod:=CTRL_MODE;

ACTION AddLogData:
Logger.s1:=INSERT('&LUX=',WORD_TO_STRING(ID),4);
IF ID<10 THEN Logger.s1:=INSERT(Logger.s1,'0',4); END_IF

//Logger.s1:=CONCAT(Logger.s1,WORD_TO_STRING(REL_V));				Logger.s1:=CONCAT(Logger.s1,';');
//Logger.s1:=CONCAT(Logger.s1,WORD_TO_STRING(REL_A));				Logger.s1:=CONCAT(Logger.s1,';');
//Logger.s1:=CONCAT(Logger.s1,DWORD_TO_STRING(ENERGYCOUNTER));	Logger.s1:=CONCAT(Logger.s1,';');

Logger.s1:=CONCAT(Logger.s1,BOOL_TO_STRING(REL_EN));			Logger.s1:=CONCAT(Logger.s1,';');	
Logger.s1:=CONCAT(Logger.s1,DWORD_TO_STRING(WORKINGTIME));		Logger.s1:=CONCAT(Logger.s1,';');
Logger.s1:=CONCAT(Logger.s1,DWORD_TO_STRING(POWERONCYCLES));	Logger.s1:=CONCAT(Logger.s1,';');

case CTRL_MODE of
	0: 	// Manuale OFF
		ModeToServer := 0;
		ForcedOn := 0;
		ForcedOff := 1;
	1:	// Manuale ON
		ModeToServer := 1;
		ForcedOn := 1;
		ForcedOff := 0;	
	2:	// Cronografo
		ModeToServer := 2;
		ForcedOn := 0;
		ForcedOff := 0;	
	3: 	//Timer 
		ModeToServer := 3;
		ForcedOn := 0;
		ForcedOff := 0;	
end_case
Logger.s1:=CONCAT(Logger.s1,BYTE_TO_STRING(ModeToServer));			Logger.s1:=CONCAT(Logger.s1,';');
Logger.s1:=CONCAT(Logger.s1,BYTE_TO_STRING(Status_Log));			Logger.s1:=CONCAT(Logger.s1,';');
Logger.s1:=CONCAT(Logger.s1,BYTE_TO_STRING(ForcedOn));			Logger.s1:=CONCAT(Logger.s1,';');
Logger.s1:=CONCAT(Logger.s1,BYTE_TO_STRING(ForcedOff));
ADDSTRING(ADR(Logger.TData), ADR(Logger.s1), Logger.TLen);
END_ACTION

ACTION StatReset:
(* Reset statistic counters *)
WORKINGTIME:=0;
POWERONCYCLES:=0;
ENERGYCOUNTER:=0;
END_ACTION

END_FUNCTION_BLOCK

// Utils Functions/FLT_TIME
FUNCTION_BLOCK FLT_TIME
VAR_INPUT
	IN		: BOOL;
	TTAP	: TIME:=T#5s;
	INITEV	: BOOL:=TRUE;
END_VAR
VAR_OUTPUT
	OUT		: BOOL;
	EVH		: BOOL;
	EVL		: BOOL;
END_VAR
VAR
	init	: BOOL:=FALSE;
	timer	: TON;
END_VAR

EVH:=FALSE;
EVL:=FALSE;

IF NOT init THEN
	init := TRUE;
	IF INITEV THEN
		OUT  := NOT IN;
	ELSE
		OUT  := IN;
	END_IF
END_IF

IF OUT<>IN THEN
	timer(IN:=TRUE,PT:=TTAP);
	IF timer.Q THEN
		OUT:=IN;
		timer(IN:=FALSE);
		IF OUT THEN EVH:=TRUE; ELSE EVL:=TRUE; END_IF
	END_IF
ELSE
	timer(IN:=FALSE);
END_IF

END_FUNCTION_BLOCK

// TCP_Logger/Logger_Proc
PROGRAM Logger_Proc
VAR
	c1:         	TCPCLIENT;

	Open:	    	BOOL;
	IpAddr:			DWORD;
	InetAddr:		DWORD;
	Connected:  	BOOL;
	Error:      	DINT;
	TxTrig:     	BOOL;
	RxData:			ARRAY [0..MAX_RECEIVE_TCP_CLIENT] OF BYTE;
	RxLen:			DINT;

	Retry:			BYTE;	(* Counter for connection retries *)
	Recovered:		BYTE;	(* Counter for recovered unsent messages *)

	i:				DINT;
	pos:			DWORD;
	hFile		: RTS_IEC_HANDLE;
	hRes		: RTS_IEC_RESULT;
	ts: STRING;
	temp	: dword;
END_VAR

(*=== State machine ===*)
CASE Logger.Status OF

	S_Logger_UNKNOWN:
		(* Startup *)
		Logger.SendReq:=FALSE;
		Open:=FALSE;
		Logger.Status:=S_Logger_IDLE;

	S_Logger_IDLE:
		(* Wait request *)
		IF Logger.SendReq THEN
			(* Resolve server name or use static IP *)
			IF LEN(Logger_SERVER)=0 THEN
				ts:=Logger_IP;
				InetAddr:=SysSockInetAddr(ts);
			ELSE
				ts:=Logger_SERVER;
				IpAddr:=SysSockGetHostByName(ts);
				DWORDSWAP(pIn:=ADR(IpAddr), pOut:=ADR(InetAddr));
			END_IF
			TxTrig:=FALSE;
			RxLen:=0;
			(* Open connection *)
			Open:=TRUE;
			Logger.Status:=S_Logger_WAITCONN;
		END_IF

	S_Logger_WAITCONN:
		(* Wait connection *)
		IF Connected THEN
			(* Send data *)
			TxTrig:=TRUE;
			Logger.Status:=S_Logger_WAITTX;
		END_IF
		IF Error>0 THEN
			Open:=FALSE;
			Logger.Status:=S_Logger_ERROR;
		END_IF

	S_Logger_WAITTX:
		(* Wait transmission *)
		IF NOT TxTrig THEN
			Logger.Status:=S_Logger_WAITRESP;
		END_IF
		IF Error>0 THEN
			Open:=FALSE;
			Logger.Status:=S_Logger_ERROR;
		END_IF

	S_Logger_WAITRESP:
		(* Wait response *)
		IF Connected=FALSE OR RxLen>=4 THEN
			Open:=FALSE;
			(* Check response *)
			IF RxLen>=4 AND CHKSTRING(pString:=ADR(RxData), pPattern:=ADR(Logger_CHECK)) THEN
				Logger.SendReq:=FALSE;
				Retry:=0;
				(* Check unsent messages to flush *)
				IF Recovered<Logger_RecoverMsgs THEN
					MsgChk();
					IF Logger.SendReq=TRUE THEN
						Recovered:=Recovered+1;
					ELSE
						Recovered:=0;
					END_IF
				ELSE
					Recovered:=0;
				END_IF
				Logger.Status:=S_Logger_IDLE;
			ELSE
				Logger.Status:=S_Logger_ERROR;
			END_IF
		END_IF

	S_Logger_ERROR:
		(* Connection error or send failure *)
		Retry:=Retry+1;
		IF Retry>Logger_ConnRetries THEN
			(* Save message as unsent *)
			MsgSave();
			Logger.SendReq:=FALSE;
			Retry:=0;
		END_IF
		Logger.Status:=S_Logger_IDLE;

ELSE
	Logger.Status:=S_Logger_UNKNOWN;
END_CASE


(*=== Execute client lib ===*)
c1(
	xOpenConnection			:= Open,
	dwInetAddr 				:= InetAddr,
	wPortNumber				:= Logger_PORT,
	ptSendData				:= ADR(Logger.SendData),
	diSendCount				:= dword_to_dint(Logger.SendLen),	// GIURE ver 4
	tConnectWatchdogTime	:= T#20S, //t#10s,
	xStartSend				:= TxTrig,
	aReceiveBuffer			:= RxData,
	diReceiveCount			:= RxLen,
	xConnected				=> Connected,
	diError					=> Error
);

(*=== Process Rx data ===*)
(*IF RxLen>0 THEN
	RxLen:=0;
END_IF*)

ACTION MsgChk:
(* Open index file *)
ts:=Logger_IndexFile;
hFile:=SysFileOpen(ts,AM_READ,ADR(hRes));
IF hFile=RTS_INVALID_HANDLE THEN
	RETURN;
END_IF
(* Search oldest message to recover *)
SysFileSetPos(hFile,Logger.LastIdxPos);
Logger.SendLen:=0;
REPEAT
	SysFileRead(hFile, ADR(Logger.SendIdx), SIZEOF(Logger.SendIdx), ADR(hRes));
	SysFileGetPos(hFile, ADR(pos));
	SysFileRead(hFile, ADR(Logger.SendLen), SIZEOF(Logger.SendLen), ADR(hRes));
	hRes:=SysFileEOF(hFile);
UNTIL
	hRes=16#0 OR Logger.SendLen<>0
END_REPEAT
SysFileClose(hFile);
(* Delete index file when all messages are recovered *)
IF Logger.SendLen=0 THEN
	Logger.LastIdxPos:=0;
	ts:=Logger_IndexFile;
	SysFileDelete(ts);
	RETURN;
END_IF
(* Recover message data *)
ts:=Logger_DataFile;
hFile:=SysFileOpen(ts,AM_READ,ADR(hRes));
IF hFile<>RTS_INVALID_HANDLE THEN
	SysFileSetPos(hFile,Logger.SendIdx);
	SysFileRead(hFile,ADR(Logger.SendData),Logger.SendLen,ADR(hRes));
	Logger.SendReq:=TRUE;
	SysFileClose(hFile);
END_IF
(* Clear index entry *)
ts:=Logger_IndexFile;
hFile:=SysFileOpen(ts,AM_READ_PLUS,ADR(hRes));
IF hFile<>RTS_INVALID_HANDLE THEN
	SysFileSetPos(hFile,pos);
	i:=0;
	SysFileWrite(hFile, ADR(i), 4, ADR(hRes));
	SysFileGetPos(hFile,ADR(Logger.LastIdxPos));
	SysFileClose(hFile);
END_IF
END_ACTION

ACTION MsgSave:
(* Add log position in recovery indexes *)
ts:=Logger_IndexFile;
hFile:=SysFileOpen(ts, AM_APPEND_PLUS, ADR(hRes));
SysFileWrite(hFile, ADR(Logger.SendIdx), SIZEOF(Logger.SendIdx), ADR(hRes));
SysFileWrite(hFile, ADR(Logger.SendLen), SIZEOF(Logger.SendLen), ADR(hRes));
SysFileClose(hFile);
END_ACTION

END_PROGRAM

// Utils Functions/DWORDSWAP
FUNCTION DWORDSWAP:BOOL
VAR_INPUT
	pIn:POINTER TO ARRAY[1..4] OF BYTE;
	pOut:POINTER TO ARRAY[1..4] OF BYTE;
END_VAR
VAR
END_VAR

pOut^[1]:=pIn^[4];
pOut^[2]:=pIn^[3];
pOut^[3]:=pIn^[2];
pOut^[4]:=pIn^[1];

END_FUNCTION

// Utils Functions/CHKSTRING
FUNCTION CHKSTRING : BOOL
VAR_INPUT
	pString: POINTER TO BYTE;
	pPattern: POINTER TO BYTE;
END_VAR
VAR
END_VAR

CHKSTRING:=TRUE;
WHILE pPattern^<>0 AND CHKSTRING DO
	IF pPattern^<>pString^ THEN CHKSTRING:=FALSE; END_IF
	pString:=pString+1;
	pPattern:=pPattern+1;
END_WHILE

END_FUNCTION

// Utils Functions/TCPCLIENT
FUNCTION_BLOCK TCPCLIENT
(***********************************************************************************************************	*)
(* Version: 1.3b                        			          													*)
(* Date: 28.10.2014                   				          							            			*)
(***********************************************************************************************************	*)
(* WAGO Kontakttechnik GmbH Hansastr. 27 32423 Minden(Westf.)													*)
(* Tel. +0049 571/887-0 Fax. +0049 571/887-0																	*)
(* Author: VB																									*)
(***********************************************************************************************************	*)
(*Description:	A TCP client to read and write data with additional connection watchdog							*)
(*History:																										*)
(*Version 1.3b: 28.10.2014: Use DWORD address for IP (Andrea Ravasio)											*)
(*Version 1.3: 11.02.2011: Changes according to 750-880/881											 			*)
(*Version 1.2: 29.08.2007 Bugfix TCP Client																		*)
(*Version 1.1: 15.01.2007 Changes according to FW11																*)
(*Version 1.0: 09.03.2006 Release																				*)
(***********************************************************************************************************	*)
VAR CONSTANT
	STATE_CREATE     				 : BYTE:= 0;
	STATE_OPEN     					 : BYTE:= 1;
	STATE_IOCTL    					 : BYTE:= 2;
	STATE_CONNECT     				 : BYTE:= 10;
	STATE_TX       					 : BYTE:= 20;
	STATE_RX       					 : BYTE:= 30;
	STATE_CLOSE    					 : BYTE:= 40;
	STATE_ERROR_TRAP			     : BYTE:= 200;
END_VAR

VAR_INPUT
	xOpenConnection					: BOOL;
	dwInetAddr						: DWORD; (* <== Use SysSockInetAddr() value or
													swapped bytes order of SysSockGetHostByName() value *)
	wPortNumber						: WORD;
	ptSendData						: POINTER TO ARRAY[0..MAX_SEND_TCP_CLIENT] OF BYTE;
	diSendCount						: DINT;
	tConnectWatchdogTime		    : TIME := t#10s;
END_VAR
VAR_OUTPUT
	xConnected						: BOOL;
	diError 						: DINT := 0;
END_VAR
(* ErrorCodes -----------------------------------------
	16#8001 => No socket descriptor available 
	16#8002 => SysSockSend returns -1 
	16#8003 => Socket was "gracefully closed" 
	16#8004 => switching to none blocking mode fails
	16#8005 => SysSockClose() returns FALSE 
    16#8006 => SysSockConnect() fails
    16#8007 => SysSockSend() fails
	16#8008 => error state machine 
	16#8009 => timeout while waiting for data from server 
------------------------------------------------------------*)
VAR_IN_OUT
	xStartSend							: BOOL;
	aReceiveBuffer						: ARRAY [0..MAX_RECEIVE_TCP_CLIENT] OF BYTE;
	diReceiveCount						: DINT;
END_VAR
VAR
	m_State								: BYTE := 0;
	m_ReceiveBuffer						: ARRAY [0..MAX_RECEIVE_TCP_CLIENT_SOCKET] OF BYTE;
	m_Socket							: DINT;
	m_AddressInfo						: SOCKADDRESS;
	m_BytesReceived						: DINT;
	m_diReturn							: DINT;
	m_xReturn							: BOOL;
	m_IoCtlParameter  					: DINT := 1; (* IOCTL-Parameter for non-blocking mode of sockets *)
	i									: INT;
	T_Connect							: TON;
	m_count								: DINT;
	diOption							: DINT := 1;
	m_Blocking   						: DINT := 0;
END_VAR

IF xOpenConnection THEN
	(* State maschine *)
	CASE  m_State OF

	(* -------------------------------------------------------------------------*)
	STATE_CREATE:
			(* create socket descriptor*)
			m_Socket := SysSockCreate(diAddressFamily	:= SOCKET_AF_INET,
													 diType		:= SOCKET_STREAM,
													 diProtocol := SOCKET_IPPROTO_TCP);
			IF m_Socket >= 0 THEN
			(*Set Push-Bit*)
				IF ADR(%MW0)=16#30000000  OR ADR(%MW0)=16#20000000 THEN (*841 or 881*)
					SysSockSetOption(
						diSocket:=m_Socket,
						diLevel:=6,
						diOption:=SOCKET_TCP_NODELAY,
						pOptionValue:=ADR(diOption),
						diOptionLength:=SIZEOF(diOption));
				ELSE
						;
				END_IF
				m_State := STATE_IOCTL; (* succesful *)
			ELSE
				diError := 16#8001;  (* no socket descriptor available *)
				m_State := STATE_ERROR_TRAP;
			END_IF

	(* -------------------------------------------------------------------------*)
	STATE_IOCTL: (* change  socket mode  to none blocking *)
		m_diReturn := SysSockIoctl( m_Socket, SOCKET_FIONBIO, ADR(m_IoCtlParameter));
		//IF m_diReturn <> 0 THEN
			m_AddressInfo.sin_family := SOCKET_AF_INET;
			m_AddressInfo.sin_port := SysSockNtohs(wPortNumber);
			m_AddressInfo.sin_addr := dwInetAddr;
			m_State := STATE_CONNECT;
		//ELSE
		//	diError := 16#8004;  (* switching to none blocking mode fails *)
		//	m_State := STATE_ERROR_TRAP;
		//END_IF


	(* -------------------------------------------------------------------------*)
	STATE_CONNECT: (* connect with server *)
		T_Connect(IN:=TRUE , PT:=tConnectWatchdogTime);(*activate watchdog for establishing connection to a server*)
		m_xReturn := SysSockConnect ( m_Socket, ADR(m_AddressInfo),  SIZEOF(m_AddressInfo));
		IF m_xReturn THEN (* succesful *)
			IF xStartSend THEN
				m_State := STATE_TX;(*transmit data*)
			ELSE
				m_State := STATE_RX;(*wait for data from server*)
			END_IF
			xConnected:=TRUE;
			T_Connect(IN:=FALSE);
		ELSE
			IF T_Connect.Q THEN
				diError := 16#8006;  (* connect fails *)
				xConnected:=FALSE;
				T_Connect(IN:=FALSE);
				m_State := STATE_ERROR_TRAP;
				SysSockClose( m_Socket);
			ELSE
				m_State := STATE_CONNECT;(*client still  tries to set up connection*)
			END_IF
		END_IF


	STATE_TX:	 (* send TCP-message *)
		m_diReturn := SysSockSend(diSocket := m_Socket,
								  pbyBuffer := ADR(ptSendData^[0]),
								  diBufferSize := diSendCount-m_count,
								  diFlags := 0);

		CASE m_diReturn OF
		-1:	(* ERROR *)
			T_Connect(IN:=TRUE , PT:=CONNECT_WATCHDOG_TIME);(*activate watchdog to check communication*)
			IF t_Connect.Q THEN
				diError := 16#8007;
				T_Connect(IN:=FALSE);
				m_State:=STATE_CLOSE;
			END_IF
		0: (* socket was "gracefully closed" *)
			m_State := STATE_CLOSE;
			diError := 16#8003;
		ELSE (* succesful *)
			m_count:=m_count+m_diReturn;
			IF m_count>=diSendCount THEN
				diError := 16#0000;
				m_State := STATE_RX;
				m_count:=0;
				xStartSend:=FALSE;
			END_IF
			T_Connect(IN:=FALSE);
		END_CASE

	(* -------------------------------------------------------------------------*)
	STATE_RX: (* process receive data *)
			m_BytesReceived := SysSockRecv(	diSocket 	:= m_Socket,
										pbyBuffer 	:= ADR(m_ReceiveBuffer),		(* Address of receive buffer *)
										diBufferSize:= SIZEOF(m_ReceiveBuffer),
										diFlags		:= 0);

			CASE m_BytesReceived OF
			-1:	(* No data available or error occured *)
				T_Connect(IN:=TRUE , PT:=tConnectWatchdogTime);(*activate watchdog to check communication*)
				IF t_Connect.Q THEN
					diError:=16#8009;
					T_Connect(IN:=FALSE);
					m_State:=STATE_CLOSE;
				END_IF
				IF xStartSend THEN
					m_State:=STATE_TX	;(* WAIT IN THIS STATE  and check for arriving data or new send command*)
				END_IF;
			0: (* socket was "gracefully closed"  *)
				m_State:=STATE_CLOSE;
				diError := 16#8003;
			ELSE (* succesful *)
				diError := 16#0000;
				T_Connect(IN:=FALSE);
				(* Copy received data into receive buffer *)
				FOR i:= 0 TO DINT_TO_INT(m_BytesReceived	)-1 DO
					aReceiveBuffer[diReceiveCount]:= m_ReceiveBuffer[i];
					diReceiveCount:=(diReceiveCount+1) MOD SIZEOF(aReceiveBuffer);
				END_FOR

			END_CASE

	(* -------------------------------------------------------------------------*)
	STATE_CLOSE : (* close socket *)
		IF ADR(%MW0)=16#30000000  OR ADR(%MW0)=16#20000000 THEN (*841 or 881*)
			;
		ELSE
			SysSockShutdown(m_Socket, 0);;(*870*)
		END_IF
		m_xReturn := SysSockClose( m_Socket);
		m_Socket := -1;
		m_State := 0; (* succesful *)
		xConnected:=FALSE;
		T_Connect(IN:=FALSE);
	(* -------------------------------------------------------------------------*)
	STATE_ERROR_TRAP: (* error handling *)
		xConnected:=FALSE;

	ELSE  (* Bad FSM code trap  *)
			m_State:= STATE_ERROR_TRAP;
			diError:= 16#8008;
	END_CASE

ELSE(*close connection*)
	IF m_Socket >= 0 THEN
		IF ADR(%MW0)=16#30000000  OR ADR(%MW0)=16#20000000 THEN (*841 or 881*)
			;
		ELSE
			SysSockShutdown(m_Socket, 0);;(*870*)
		END_IF
		SysSockClose( m_Socket);
	END_IF
	m_Socket := -1;
	diError := 16#0000;
	m_State := STATE_CREATE;
	xConnected:=FALSE;
	T_Connect(IN:=FALSE);
END_IF

END_FUNCTION_BLOCK

// TCP_Remote/Remote_Proc
PROGRAM Remote_Proc
VAR
	s1:         	TCPSERVER;
	Enable: 		BOOL;
	Connected: 		BOOL;
	Error: 			DINT;

	TxData:			ARRAY [0..MAX_SEND_TCP_SERVER] OF BYTE;
	TxLen:			DINT;
	TxTrig:			BOOL;

	RxData:			ARRAY [0..MAX_RECEIVE_TCP_SERVER] OF BYTE;
	RxLen:			DINT;

	Status:			DINT;

	(* Command interpreter *)

	Cmd_Buf:		ARRAY [0..MAX_RECEIVE_TCP_SERVER] OF BYTE;
	Cmd_Buf_U16:	POINTER TO WORD;
	Cmd_Buf_INT:	POINTER TO INT;
	Cmd_BufLen:		WORD;
	Cmd_St:			WORD;

	Cmd_Obj:		WORD;
	Cmd_ObjIdx:		WORD;
	Cmd_C:			WORD;
	Cmd_R:			WORD;
	Cmd_CLen:		WORD;
	Cmd_RLen:		WORD;

	i : WORD;
	j : INT;
	s2 : STRING;
	x : word;
	NewValueTimer: dword;

	Result: bool;
	DateTime: DT;
	DTStr: string;
	Year: word;
	Month, Day, Hour, minute, Sec: byte;
	LocalSetpoint: array[0..95] of word;
	Plant_SN_H_W, Plant_SN_L_W:	word;
	Plant_SN_H, Plant_SN_L: dword;
	NewValueTimerH, NewValueTimerL: word;
	ModeFromPlc	: word;
END_VAR

(*=== State machine ===*)
CASE Status OF
	0: (* Startup *)
		TxLen:=0; TxTrig:=FALSE;
		RxLen:=0;
		Enable:=TRUE;
		Status:=1;

	1: (* Wait incoming connection *)
		IF Connected THEN
			(* Log access *)
			//LogEv(EL_Log,EO_VPN,1,5,'Remote');
			(* Send welcome message *)
			(*ADDSTRING(pTxData:=ADR(TxData), pString:=ADR(Remote_WELCOME), TxLen:=TxLen);
			TxTrig:=TRUE;*)
			(* Reset vars *)
			Cmd_BufLen:=0;
			Cmd_St:=0;
			Status:=2;
		END_IF
		IF Error>1 THEN
			Enable:=FALSE;
			Status:=0;
		END_IF

	2: (* Wait command *)
		IF RxLen>0 THEN
			(*=== Interpreter start ===*)
			IF Cmd_BufLen+(RxLen/2)>=MAX_RECEIVE_TCP_SERVER THEN
				(* ERROR *)
				Cmd_BufLen:=0;
			ELSE
				i:=HEXTORAW(pString:=ADR(RxData), StringLen:=DINT_TO_WORD(RxLen), pData:=ADR(Cmd_Buf[Cmd_BufLen]));
				Cmd_BufLen:=Cmd_BufLen+i;
			END_IF
			IF Cmd_BufLen>=8 THEN
				Cmd_Buf_U16:=ADR(Cmd_Buf[6]);
					(* Log command *)
				IF Cmd_BufLen>=(8+byte_to_word(Cmd_Buf[6])) THEN	
					Cmd_Obj:=byte_to_word(Cmd_Buf[0]);
					Cmd_ObjIdx:=byte_to_word(Cmd_Buf[3]); //memorizzo il byte più significativo (yy) di |xxyy|
					Cmd_ObjIdx:=SHL(Cmd_ObjIdx,8); //shift a sx di 8 bit
					Cmd_ObjIdx:=Cmd_ObjIdx+byte_to_word(Cmd_Buf[2]); //aggiungo il byte meno significativo (xx)
					Cmd_C:=byte_to_word(Cmd_Buf[4]);
					Cmd_CLen:=byte_to_word(Cmd_Buf[6]);
					(* Execute command *)
					Command();
					Cmd_BufLen:=0;
				END_IF
			END_IF
			(*=== Interpreter end ===*)
			RxLen:=0;
		END_IF
		IF NOT Connected THEN
			Status:=0;
		END_IF

ELSE
	Status:=0;
END_CASE


(*=== Execute server lib ===*)
s1(
	xEnable				:= Enable,
	wPortNumber			:= Remote_PORT,
	tServerTimeOut		:= t#10s,//t#15m,
	ptSendData			:= ADR(TxData),
	diSendCount			:= TxLen,
	xStartSend			:= TxTrig,
	aReceiveBuffer		:= RxData,
	diReceiveCount		:= RxLen,
	xClientConnected	=> Connected,
	diError				=> Error
);

ACTION Cmd_CAL:
(* Check index *)
IF Cmd_ObjIdx<1 OR Cmd_ObjIdx>17 THEN
	Cmd_R:=2;
	RETURN;
END_IF

(* Process command *)
CASE Cmd_C OF

	1: (* TRY REARM *)

	
ELSE
	Cmd_R:=3;
END_CASE
END_ACTION

ACTION Cmd_CRON:
(* Check index *)
if Cmd_ObjIdx<1 OR Cmd_ObjIdx>MAX_LUXNUM then
	Cmd_R:=2;
	return;
end_if

